LIN {X 0,Y 203.448,Z 428.589,A -85,B 0,C 180,E1 -22081.79,E2 -22081.79} C_VEL
LIN {X 0,Y 207.049,Z 418.268,A -85,B 0,C 180,E1 -22083.768,E2 -22083.768} C_VEL
LIN {X 0,Y 210.594,Z 406.82,A -85,B 0,C 180,E1 -22085.44,E2 -22085.44} C_VEL
LIN {X 0,Y 213.533,Z 394.846,A -85,B 0,C 180,E1 -22086.77,E2 -22086.77} C_VEL
LIN {X 0,Y 215.971,Z 381.541,A -85,B 0,C 180,E1 -22087.821,E2 -22087.821} C_VEL
LIN {X 0,Y 217.695,Z 368.318,A -85,B 0,C 180,E1 -22088.489,E2 -22088.489} C_VEL
LIN {X 0,Y 220.282,Z 324.105,A -85,B 0,C 180,E1 -22089.842,E2 -22089.842} C_VEL
LIN {X 0,Y 219.565,Z 319.298,A -85,B 0,C 180,E1 -22090.222,E2 -22090.222} C_VEL
LIN {X 0,Y 213.219,Z 304.183,A -85,B 0,C 180,E1 -22092.522,E2 -22092.522} C_VEL
LIN {X 0,Y 207.872,Z 293.408,A -85,B 0,C 180,E1 -22094.554,E2 -22094.554} C_VEL
LIN {X 0,Y 202.404,Z 283.572,A -85,B 0,C 180,E1 -22096.771,E2 -22096.771} C_VEL
LIN {X 0,Y 197.273,Z 275.162,A -85,B 0,C 180,E1 -22099.019,E2 -22099.019} C_VEL
LIN {X 0,Y 193.69,Z 269.753,A -85,B 0,C 180,E1 -22100.705,E2 -22100.705} C_VEL
LIN {X 0,Y 190.17,Z 264.45,A -85,B 0,C 180,E1 -22102.496,E2 -22102.496} C_VEL
LIN {X 0,Y 187.207,Z 260.568,A -85,B 0,C 180,E1 -22104.085,E2 -22104.085} C_VEL
LIN {X 0,Y 186.277,Z 258.764,A -85,B 0,C 180,E1 -22104.71,E2 -22104.71} C_VEL
LIN {X 0,Y 185.559,Z 256.36,A -85,B 0,C 180,E1 -22107.046,E2 -22107.046} C_VEL
LIN {X 0,Y 185.548,Z 256.361,A -85,B 0,C 180,E1 -22110.595,E2 -22110.595} C_VEL
LIN {X 0,Y 185.581,Z 256.359,A -85,B 0,C 180,E1 -22115.382,E2 -22115.382} C_VEL
LIN {X 0,Y 185.635,Z 256.363,A -85,B 0,C 180,E1 -22121.171,E2 -22121.171} C_VEL
LIN {X 0,Y 185.673,Z 256.35,A -85,B 0,C 180,E1 -22124.636,E2 -22124.636} C_VEL
LIN {X 0,Y 185.925,Z 256.316,A -85,B 0,C 180,E1 -22129.359,E2 -22129.359} C_VEL
LIN {X 0,Y 185.958,Z 256.306,A -85,B 0,C 180,E1 -22133.49,E2 -22133.49} C_VEL
LIN {X 0,Y 186.203,Z 256.274,A -85,B 0,C 180,E1 -22137.837,E2 -22137.837} C_VEL
LIN {X 0,Y 186.405,Z 256.262,A -85,B 0,C 180,E1 -22140,E2 -22140} C_VEL
LIN {X 0,Y 185.909,Z 256.317,A -85,B 0,C 180,E1 -22144.336,E2 -22144.336} C_VEL
LIN {X 0,Y 185.976,Z 256.304,A -85,B 0,C 180,E1 -22148.694,E2 -22148.694} C_VEL
LIN {X 0,Y 185.724,Z 256.336,A -85,B 0,C 180,E1 -22153.124,E2 -22153.124} C_VEL
LIN {X 0,Y 185.688,Z 256.34,A -85,B 0,C 180,E1 -22157.625,E2 -22157.625} C_VEL
LIN {X 0,Y 185.597,Z 256.352,A -85,B 0,C 180,E1 -22162.252,E2 -22162.252} C_VEL
LIN {X 0,Y 185.564,Z 256.36,A -85,B 0,C 180,E1 -22167.032,E2 -22167.032} C_VEL
LIN {X 0,Y 185.607,Z 256.374,A -85,B 0,C 180,E1 -22169.284,E2 -22169.284} C_VEL
LIN {X 0,Y 186.334,Z 258.759,A -85,B 0,C 180,E1 -22169.804,E2 -22169.804} C_VEL
LIN {X 0,Y 188.069,Z 260.918,A -85,B 0,C 180,E1 -22170.763,E2 -22170.763} C_VEL
LIN {X 0,Y 189.675,Z 262.213,A -85,B 0,C 180,E1 -22171.569,E2 -22171.569} C_VEL
LIN {X 0,Y 191.536,Z 265.32,A -85,B 0,C 180,E1 -22172.568,E2 -22172.568} C_VEL
LIN {X 0,Y 193.597,Z 267.452,A -85,B 0,C 180,E1 -22173.544,E2 -22173.544} C_VEL
LIN {X 0,Y 196.036,Z 270.879,A -85,B 0,C 180,E1 -22174.698,E2 -22174.698} C_VEL
LIN {X 0,Y 197.873,Z 273.45,A -85,B 0,C 180,E1 -22175.528,E2 -22175.528} C_VEL
LIN {X 0,Y 200.738,Z 277.395,A -85,B 0,C 180,E1 -22176.761,E2 -22176.761} C_VEL
LIN {X 0,Y 206.923,Z 286.536,A -85,B 0,C 180,E1 -22179.242,E2 -22179.242} C_VEL
LIN {X 0,Y 210.932,Z 293.337,A -85,B 0,C 180,E1 -22180.757,E2 -22180.757} C_VEL
LIN {X 0,Y 217.361,Z 306.275,A -85,B 0,C 180,E1 -22183.082,E2 -22183.082} C_VEL
LIN {X 0,Y 220.832,Z 314.289,A -85,B 0,C 180,E1 -22184.29,E2 -22184.29} C_VEL
LIN {X 0,Y 218.061,Z 360.113,A -85,B 0,C 180,E1 -22185.691,E2 -22185.691} C_VEL
LIN {X 0,Y 216.493,Z 373.353,A -85,B 0,C 180,E1 -22186.429,E2 -22186.429} C_VEL
LIN {X 0,Y 214.306,Z 385.674,A -85,B 0,C 180,E1 -22187.438,E2 -22187.438} C_VEL
LIN {X 0,Y 211.711,Z 396.969,A -85,B 0,C 180,E1 -22188.717,E2 -22188.717} C_VEL
LIN {X 0,Y 208.24,Z 408.631,A -85,B 0,C 180,E1 -22190.43,E2 -22190.43} C_VEL
LIN {X 0,Y 204.695,Z 419.107,A -85,B 0,C 180,E1 -22192.452,E2 -22192.452} C_VEL
LIN {X 0,Y 200.989,Z 428.49,A -85,B 0,C 180,E1 -22194.763,E2 -22194.763} C_VEL
LIN {X 0,Y 197.612,Z 436.177,A -85,B 0,C 180,E1 -22197.155,E2 -22197.155} C_VEL
LIN {X 0,Y 193.935,Z 444.033,A -85,B 0,C 180,E1 -22200.298,E2 -22200.298} C_VEL
LIN {X 0,Y 190.616,Z 450.593,A -85,B 0,C 180,E1 -22203.74,E2 -22203.74} C_VEL
LIN {X 0,Y 188.133,Z 455.122,A -85,B 0,C 180,E1 -22206.906,E2 -22206.906} C_VEL
LIN {X 0,Y 185.771,Z 459.292,A -85,B 0,C 180,E1 -22211.049,E2 -22211.049} C_VEL
LIN {X 0,Y 184.359,Z 461.532,A -85,B 0,C 180,E1 -22214.523,E2 -22214.523} C_VEL
LIN {X 0,Y 183.67,Z 462.424,A -85,B 0,C 180,E1 -22216.727,E2 -22216.727} C_VEL
LIN {X 0,Y 183.286,Z 462.899,A -85,B 0,C 180,E1 -22218.947,E2 -22218.947} C_VEL
LIN {X 0,Y 183.106,Z 462.953,A -85,B 0,C 180,E1 -22221.168,E2 -22221.168} C_VEL
LIN {X 0,Y 183.082,Z 462.624,A -85,B 0,C 180,E1 -22223.387,E2 -22223.387} C_VEL
LIN {X 0,Y 183.132,Z 461.645,A -85,B 0,C 180,E1 -22226.201,E2 -22226.201} C_VEL
LIN {X 0,Y 183.433,Z 459.249,A -85,B 0,C 180,E1 -22230,E2 -22230} C_VEL
LIN {X 0,Y 184.027,Z 456.15,A -85,B 0,C 180,E1 -22233.284,E2 -22233.284} C_VEL
LIN {X 0,Y 184.978,Z 452.007,A -85,B 0,C 180,E1 -22236.545,E2 -22236.545} C_VEL
LIN {X 0,Y 186.753,Z 445.691,A -85,B 0,C 180,E1 -22240.297,E2 -22240.297} C_VEL
LIN {X 0,Y 188.757,Z 438.816,A -85,B 0,C 180,E1 -22243.456,E2 -22243.456} C_VEL
LIN {X 0,Y 191.319,Z 430.194,A -85,B 0,C 180,E1 -22246.54,E2 -22246.54} C_VEL
LIN {X 0,Y 193.755,Z 421.37,A -85,B 0,C 180,E1 -22249.054,E2 -22249.054} C_VEL
LIN {X 0,Y 196.263,Z 411.56,A -85,B 0,C 180,E1 -22251.285,E2 -22251.285} C_VEL
LIN {X 0,Y 198.602,Z 401.054,A -85,B 0,C 180,E1 -22253.184,E2 -22253.184} C_VEL
LIN {X 0,Y 200.825,Z 389.158,A -85,B 0,C 180,E1 -22254.831,E2 -22254.831} C_VEL
LIN {X 0,Y 202.636,Z 376.778,A -85,B 0,C 180,E1 -22256.106,E2 -22256.106} C_VEL
LIN {X 0,Y 203.926,Z 363.965,A -85,B 0,C 180,E1 -22257.031,E2 -22257.031} C_VEL
LIN {X 0,Y 204.857,Z 349.414,A -85,B 0,C 180,E1 -22257.622,E2 -22257.622} C_VEL
LIN {X 0,Y 207.063,Z 299.532,A -85,B 0,C 180,E1 -22259.251,E2 -22259.251} C_VEL
LIN {X 0,Y 200.953,Z 283.961,A -85,B 0,C 180,E1 -22261.036,E2 -22261.036} C_VEL
LIN {X 0,Y 195.353,Z 273.341,A -85,B 0,C 180,E1 -22262.644,E2 -22262.644} C_VEL
LIN {X 0,Y 189.717,Z 264.038,A -85,B 0,C 180,E1 -22264.328,E2 -22264.328} C_VEL
LIN {X 0,Y 187.441,Z 260.424,A -85,B 0,C 180,E1 -22265.042,E2 -22265.042} C_VEL
LIN {X 0,Y 185.812,Z 257.687,A -85,B 0,C 180,E1 -22265.575,E2 -22265.575} C_VEL
LIN {X 0,Y 185.526,Z 256.374,A -85,B 0,C 180,E1 -22265.765,E2 -22265.765} C_VEL
LIN {X 0,Y 185.473,Z 256.381,A -85,B 0,C 180,E1 -22270.725,E2 -22270.725} C_VEL
LIN {X 0,Y 185.463,Z 256.382,A -85,B 0,C 180,E1 -22276.054,E2 -22276.054} C_VEL
LIN {X 0,Y 185.47,Z 256.382,A -85,B 0,C 180,E1 -22279.895,E2 -22279.895} C_VEL
LIN {X 0,Y 185.508,Z 256.377,A -85,B 0,C 180,E1 -22282.711,E2 -22282.711} C_VEL
LIN {X 0,Y 185.543,Z 256.343,A -85,B 0,C 180,E1 -22287.974,E2 -22287.974} C_VEL
LIN {X 0,Y 185.582,Z 256.359,A -85,B 0,C 180,E1 -22290.576,E2 -22290.576} C_VEL
LIN {X 0,Y 185.589,Z 256.348,A -85,B 0,C 180,E1 -22295.382,E2 -22295.382} C_VEL
LIN {X 0,Y 185.676,Z 256.346,A -85,B 0,C 180,E1 -22301.133,E2 -22301.133} C_VEL
LIN {X 0,Y 185.696,Z 256.345,A -85,B 0,C 180,E1 -22304.637,E2 -22304.637} C_VEL
LIN {X 0,Y 185.889,Z 256.288,A -85,B 0,C 180,E1 -22309.419,E2 -22309.419} C_VEL
LIN {X 0,Y 185.938,Z 256.318,A -85,B 0,C 180,E1 -22313.489,E2 -22313.489} C_VEL
LIN {X 0,Y 186.204,Z 256.277,A -85,B 0,C 180,E1 -22317.837,E2 -22317.837} C_VEL
LIN {X 0,Y 186.405,Z 256.262,A -85,B 0,C 180,E1 -22320,E2 -22320} C_VEL
LIN {X 0,Y 185.923,Z 256.315,A -85,B 0,C 180,E1 -22324.336,E2 -22324.336} C_VEL
LIN {X 0,Y 186.03,Z 256.307,A -85,B 0,C 180,E1 -22328.691,E2 -22328.691} C_VEL
LIN {X 0,Y 185.726,Z 256.342,A -85,B 0,C 180,E1 -22333.123,E2 -22333.123} C_VEL
LIN {X 0,Y 185.657,Z 256.347,A -85,B 0,C 180,E1 -22337.628,E2 -22337.628} C_VEL
LIN {X 0,Y 185.571,Z 256.37,A -85,B 0,C 180,E1 -22342.254,E2 -22342.254} C_VEL
LIN {X 0,Y 185.577,Z 256.357,A -85,B 0,C 180,E1 -22344.646,E2 -22344.646} C_VEL
LIN {X 0,Y 185.544,Z 256.367,A -85,B 0,C 180,E1 -22349.499,E2 -22349.499} C_VEL
LIN {X 0,Y 185.497,Z 256.372,A -85,B 0,C 180,E1 -22354.632,E2 -22354.632} C_VEL
LIN {X 0,Y 185.501,Z 256.378,A -85,B 0,C 180,E1 -22357.314,E2 -22357.314} C_VEL
LIN {X 0,Y 185.464,Z 256.384,A -85,B 0,C 180,E1 -22360.722,E2 -22360.722} C_VEL
LIN {X 0,Y 185.47,Z 256.406,A -85,B 0,C 180,E1 -22366.098,E2 -22366.098} C_VEL
LIN {X 0,Y 186.5,Z 260.261,A -85,B 0,C 180,E1 -22368.365,E2 -22368.365} C_VEL
LIN {X 0,Y 188.973,Z 264.686,A -85,B 0,C 180,E1 -22369.172,E2 -22369.172} C_VEL
LIN {X 0,Y 195.749,Z 278.235,A -85,B 0,C 180,E1 -22371.304,E2 -22371.304} C_VEL
LIN {X 0,Y 202.24,Z 293.675,A -85,B 0,C 180,E1 -22373.268,E2 -22373.268} C_VEL
LIN {X 0,Y 204.621,Z 300.449,A -85,B 0,C 180,E1 -22373.993,E2 -22373.993} C_VEL
LIN {X 0,Y 206.416,Z 317.831,A -85,B 0,C 180,E1 -22375.02,E2 -22375.02} C_VEL
LIN {X 0,Y 206.011,Z 326.955,A -85,B 0,C 180,E1 -22375.317,E2 -22375.317} C_VEL
LIN {X 0,Y 205.217,Z 332.797,A -85,B 0,C 180,E1 -22375.416,E2 -22375.416} C_VEL
LIN {X 0,Y 199.436,Z 351.769,A -85,B 0,C 180,E1 -22375.178,E2 -22375.178} C_VEL
LIN {X 0,Y 198.574,Z 357.613,A -85,B 0,C 180,E1 -22375.267,E2 -22375.267} C_VEL
LIN {X 0,Y 197.647,Z 372.415,A -85,B 0,C 180,E1 -22375.864,E2 -22375.864} C_VEL
LIN {X 0,Y 196.156,Z 385.164,A -85,B 0,C 180,E1 -22376.727,E2 -22376.727} C_VEL
LIN {X 0,Y 194.021,Z 397.941,A -85,B 0,C 180,E1 -22378.011,E2 -22378.011} C_VEL
LIN {X 0,Y 191.532,Z 410.148,A -85,B 0,C 180,E1 -22379.7,E2 -22379.7} C_VEL
LIN {X 0,Y 188.837,Z 421.006,A -85,B 0,C 180,E1 -22381.672,E2 -22381.672} C_VEL
LIN {X 0,Y 185.792,Z 431.841,A -85,B 0,C 180,E1 -22384.214,E2 -22384.214} C_VEL
LIN {X 0,Y 183.265,Z 441.005,A -85,B 0,C 180,E1 -22386.981,E2 -22386.981} C_VEL
LIN {X 0,Y 181.313,Z 447.926,A -85,B 0,C 180,E1 -22389.583,E2 -22389.583} C_VEL
LIN {X 0,Y 179.202,Z 455.049,A -85,B 0,C 180,E1 -22392.894,E2 -22392.894} C_VEL
LIN {X 0,Y 177.601,Z 460.726,A -85,B 0,C 180,E1 -22396.265,E2 -22396.265} C_VEL
LIN {X 0,Y 176.675,Z 465.196,A -85,B 0,C 180,E1 -22399.688,E2 -22399.688} C_VEL
LIN {X 0,Y 176.137,Z 468.572,A -85,B 0,C 180,E1 -22403.125,E2 -22403.125} C_VEL
LIN {X 0,Y 175.995,Z 471.007,A -85,B 0,C 180,E1 -22406.681,E2 -22406.681} C_VEL
LIN {X 0,Y 176.092,Z 472.381,A -85,B 0,C 180,E1 -22410,E2 -22410} C_VEL
LIN {X 0,Y 175.97,Z 472.854,A -85,B 0,C 180,E1 -22413.176,E2 -22413.176} C_VEL
LIN {X 0,Y 176.141,Z 472.465,A -85,B 0,C 180,E1 -22416.875,E2 -22416.875} C_VEL
LIN {X 0,Y 176.481,Z 471.725,A -85,B 0,C 180,E1 -22419.166,E2 -22419.166} C_VEL
LIN {X 0,Y 177.064,Z 470.558,A -85,B 0,C 180,E1 -22421.447,E2 -22421.447} C_VEL
LIN {X 0,Y 177.887,Z 468.974,A -85,B 0,C 180,E1 -22423.713,E2 -22423.713} C_VEL
LIN {X 0,Y 179.541,Z 465.81,A -85,B 0,C 180,E1 -22427.073,E2 -22427.073} C_VEL
LIN {X 0,Y 181.936,Z 461.603,A -85,B 0,C 180,E1 -22430.344,E2 -22430.344} C_VEL
LIN {X 0,Y 185.407,Z 455.225,A -85,B 0,C 180,E1 -22434.047,E2 -22434.047} C_VEL
LIN {X 0,Y 188.77,Z 448.292,A -85,B 0,C 180,E1 -22437.134,E2 -22437.134} C_VEL
LIN {X 0,Y 192.793,Z 439.621,A -85,B 0,C 180,E1 -22440.082,E2 -22440.082} C_VEL
LIN {X 0,Y 196.671,Z 430.752,A -85,B 0,C 180,E1 -22442.413,E2 -22442.413} C_VEL
LIN {X 0,Y 200.782,Z 419.841,A -85,B 0,C 180,E1 -22444.667,E2 -22444.667} C_VEL
LIN {X 0,Y 204.401,Z 408.803,A -85,B 0,C 180,E1 -22446.378,E2 -22446.378} C_VEL
LIN {X 0,Y 207.665,Z 396.448,A -85,B 0,C 180,E1 -22447.836,E2 -22447.836} C_VEL
LIN {X 0,Y 210.073,Z 384.716,A -85,B 0,C 180,E1 -22448.85,E2 -22448.85} C_VEL
LIN {X 0,Y 211.952,Z 371.86,A -85,B 0,C 180,E1 -22449.599,E2 -22449.599} C_VEL
LIN {X 0,Y 213.178,Z 357.263,A -85,B 0,C 180,E1 -22450.1,E2 -22450.1} C_VEL
LIN {X 0,Y 214.965,Z 324.362,A -85,B 0,C 180,E1 -22451.136,E2 -22451.136} C_VEL
LIN {X 0,Y 214.444,Z 321.886,A -85,B 0,C 180,E1 -22451.382,E2 -22451.382} C_VEL
LIN {X 0,Y 208.578,Z 307.84,A -85,B 0,C 180,E1 -22453.637,E2 -22453.637} C_VEL
LIN {X 0,Y 203.693,Z 297.749,A -85,B 0,C 180,E1 -22455.61,E2 -22455.61} C_VEL
LIN {X 0,Y 198.733,Z 288.663,A -85,B 0,C 180,E1 -22457.736,E2 -22457.736} C_VEL
LIN {X 0,Y 193.493,Z 279.929,A -85,B 0,C 180,E1 -22460.167,E2 -22460.167} C_VEL
LIN {X 0,Y 190.645,Z 275.459,A -85,B 0,C 180,E1 -22461.59,E2 -22461.59} C_VEL
LIN {X 0,Y 186.999,Z 269.999,A -85,B 0,C 180,E1 -22463.539,E2 -22463.539} C_VEL
LIN {X 0,Y 183.891,Z 265.461,A -85,B 0,C 180,E1 -22465.339,E2 -22465.339} C_VEL
LIN {X 0,Y 179.125,Z 259.472,A -85,B 0,C 180,E1 -22468.347,E2 -22468.347} C_VEL
LIN {X 0,Y 178.697,Z 258.346,A -85,B 0,C 180,E1 -22468.758,E2 -22468.758} C_VEL
LIN {X 0,Y 178.482,Z 257.241,A -85,B 0,C 180,E1 -22470.03,E2 -22470.03} C_VEL
LIN {X 0,Y 178.516,Z 257.237,A -85,B 0,C 180,E1 -22474.889,E2 -22474.889} C_VEL
LIN {X 0,Y 178.591,Z 257.239,A -85,B 0,C 180,E1 -22480.814,E2 -22480.814} C_VEL
LIN {X 0,Y 178.651,Z 257.227,A -85,B 0,C 180,E1 -22486.347,E2 -22486.347} C_VEL
LIN {X 0,Y 178.961,Z 257.19,A -85,B 0,C 180,E1 -22490.962,E2 -22490.962} C_VEL
LIN {X 0,Y 179.149,Z 257.153,A -85,B 0,C 180,E1 -22497.752,E2 -22497.752} C_VEL
LIN {X 0,Y 179.368,Z 257.138,A -85,B 0,C 180,E1 -22500,E2 -22500} C_VEL
LIN {X 0,Y 178.857,Z 257.196,A -85,B 0,C 180,E1 -22504.508,E2 -22504.508} C_VEL
LIN {X 0,Y 178.906,Z 257.186,A -85,B 0,C 180,E1 -22509.041,E2 -22509.041} C_VEL
LIN {X 0,Y 178.653,Z 257.216,A -85,B 0,C 180,E1 -22513.653,E2 -22513.653} C_VEL
LIN {X 0,Y 178.624,Z 257.223,A -85,B 0,C 180,E1 -22519.216,E2 -22519.216} C_VEL
LIN {X 0,Y 178.534,Z 257.239,A -85,B 0,C 180,E1 -22525.274,E2 -22525.274} C_VEL
LIN {X 0,Y 178.539,Z 257.332,A -85,B 0,C 180,E1 -22525.562,E2 -22525.562} C_VEL
LIN {X 0,Y 179.259,Z 259.662,A -85,B 0,C 180,E1 -22526.172,E2 -22526.172} C_VEL
LIN {X 0,Y 181.191,Z 261.941,A -85,B 0,C 180,E1 -22527.427,E2 -22527.427} C_VEL
LIN {X 0,Y 182.827,Z 263.049,A -85,B 0,C 180,E1 -22528.373,E2 -22528.373} C_VEL
LIN {X 0,Y 184.655,Z 266.207,A -85,B 0,C 180,E1 -22529.518,E2 -22529.518} C_VEL
LIN {X 0,Y 186.908,Z 268.442,A -85,B 0,C 180,E1 -22530.74,E2 -22530.74} C_VEL
LIN {X 0,Y 189.389,Z 271.993,A -85,B 0,C 180,E1 -22532.082,E2 -22532.082} C_VEL
LIN {X 0,Y 190.753,Z 273.562,A -85,B 0,C 180,E1 -22532.762,E2 -22532.762} C_VEL
LIN {X 0,Y 194.542,Z 278.861,A -85,B 0,C 180,E1 -22534.601,E2 -22534.601} C_VEL
LIN {X 0,Y 199.477,Z 285.887,A -85,B 0,C 180,E1 -22536.795,E2 -22536.795} C_VEL
LIN {X 0,Y 205.61,Z 295.649,A -85,B 0,C 180,E1 -22539.303,E2 -22539.303} C_VEL
LIN {X 0,Y 211.796,Z 308.073,A -85,B 0,C 180,E1 -22541.701,E2 -22541.701} C_VEL
LIN {X 0,Y 215.496,Z 316.487,A -85,B 0,C 180,E1 -22543.069,E2 -22543.069} C_VEL
LIN {X 0,Y 212.733,Z 360.615,A -85,B 0,C 180,E1 -22544.451,E2 -22544.451} C_VEL
LIN {X 0,Y 211.091,Z 373.864,A -85,B 0,C 180,E1 -22545.206,E2 -22545.206} C_VEL
LIN {X 0,Y 208.85,Z 385.963,A -85,B 0,C 180,E1 -22546.215,E2 -22546.215} C_VEL
LIN {X 0,Y 205.925,Z 398.03,A -85,B 0,C 180,E1 -22547.62,E2 -22547.62} C_VEL
LIN {X 0,Y 202.321,Z 409.533,A -85,B 0,C 180,E1 -22549.36,E2 -22549.36} C_VEL
LIN {X 0,Y 198.799,Z 419.507,A -85,B 0,C 180,E1 -22551.344,E2 -22551.344} C_VEL
LIN {X 0,Y 195.169,Z 428.309,A -85,B 0,C 180,E1 -22553.547,E2 -22553.547} C_VEL
LIN {X 0,Y 191.584,Z 436.061,A -85,B 0,C 180,E1 -22555.984,E2 -22555.984} C_VEL
LIN {X 0,Y 187.589,Z 444.231,A -85,B 0,C 180,E1 -22559.329,E2 -22559.329} C_VEL
LIN {X 0,Y 184.177,Z 450.592,A -85,B 0,C 180,E1 -22562.748,E2 -22562.748} C_VEL
LIN {X 0,Y 181.538,Z 455.17,A -85,B 0,C 180,E1 -22566.015,E2 -22566.015} C_VEL
LIN {X 0,Y 179.44,Z 458.636,A -85,B 0,C 180,E1 -22569.36,E2 -22569.36} C_VEL
LIN {X 0,Y 178.349,Z 460.36,A -85,B 0,C 180,E1 -22571.624,E2 -22571.624} C_VEL
LIN {X 0,Y 177.433,Z 461.666,A -85,B 0,C 180,E1 -22573.903,E2 -22573.903} C_VEL
LIN {X 0,Y 176.248,Z 463.086,A -85,B 0,C 180,E1 -22578.499,E2 -22578.499} C_VEL
LIN {X 0,Y 176.025,Z 463.16,A -85,B 0,C 180,E1 -22580.81,E2 -22580.81} C_VEL
LIN {X 0,Y 175.973,Z 462.849,A -85,B 0,C 180,E1 -22583.119,E2 -22583.119} C_VEL
LIN {X 0,Y 176.044,Z 461.72,A -85,B 0,C 180,E1 -22586.426,E2 -22586.426} C_VEL
LIN {X 0,Y 176.344,Z 459.547,A -85,B 0,C 180,E1 -22590,E2 -22590} C_VEL
LIN {X 0,Y 176.97,Z 456.487,A -85,B 0,C 180,E1 -22593.415,E2 -22593.415} C_VEL
LIN {X 0,Y 177.957,Z 452.386,A -85,B 0,C 180,E1 -22596.804,E2 -22596.804} C_VEL
LIN {X 0,Y 179.796,Z 446.116,A -85,B 0,C 180,E1 -22600.7,E2 -22600.7} C_VEL
LIN {X 0,Y 181.895,Z 439.295,A -85,B 0,C 180,E1 -22603.974,E2 -22603.974} C_VEL
LIN {X 0,Y 184.563,Z 430.76,A -85,B 0,C 180,E1 -22607.164,E2 -22607.164} C_VEL
LIN {X 0,Y 187.088,Z 422.011,A -85,B 0,C 180,E1 -22609.76,E2 -22609.76} C_VEL
LIN {X 0,Y 189.92,Z 411.473,A -85,B 0,C 180,E1 -22612.233,E2 -22612.233} C_VEL
LIN {X 0,Y 192.466,Z 400.411,A -85,B 0,C 180,E1 -22614.255,E2 -22614.255} C_VEL
LIN {X 0,Y 194.807,Z 388.28,A -85,B 0,C 180,E1 -22615.94,E2 -22615.94} C_VEL
LIN {X 0,Y 196.662,Z 375.572,A -85,B 0,C 180,E1 -22617.25,E2 -22617.25} C_VEL
LIN {X 0,Y 197.989,Z 362.526,A -85,B 0,C 180,E1 -22618.147,E2 -22618.147} C_VEL
LIN {X 0,Y 199.089,Z 343.717,A -85,B 0,C 180,E1 -22618.867,E2 -22618.867} C_VEL
LIN {X 0,Y 201.058,Z 301.314,A -85,B 0,C 180,E1 -22620.281,E2 -22620.281} C_VEL
LIN {X 0,Y 195.021,Z 286.063,A -85,B 0,C 180,E1 -22622.148,E2 -22622.148} C_VEL
LIN {X 0,Y 187.68,Z 272.688,A -85,B 0,C 180,E1 -22624.399,E2 -22624.399} C_VEL
LIN {X 0,Y 180.717,Z 261.583,A -85,B 0,C 180,E1 -22626.697,E2 -22626.697} C_VEL
LIN {X 0,Y 179.059,Z 259.332,A -85,B 0,C 180,E1 -22627.262,E2 -22627.262} C_VEL
LIN {X 0,Y 178.448,Z 257.256,A -85,B 0,C 180,E1 -22627.622,E2 -22627.622} C_VEL
LIN {X 0,Y 178.4,Z 257.26,A -85,B 0,C 180,E1 -22632.044,E2 -22632.044} C_VEL
LIN {X 0,Y 178.396,Z 257.262,A -85,B 0,C 180,E1 -22635.163,E2 -22635.163} C_VEL
LIN {X 0,Y 178.405,Z 257.261,A -85,B 0,C 180,E1 -22638.458,E2 -22638.458} C_VEL
LIN {X 0,Y 178.424,Z 257.259,A -85,B 0,C 180,E1 -22643.783,E2 -22643.783} C_VEL
LIN {X 0,Y 178.487,Z 257.226,A -85,B 0,C 180,E1 -22646.546,E2 -22646.546} C_VEL
LIN {X 0,Y 178.523,Z 257.234,A -85,B 0,C 180,E1 -22650.007,E2 -22650.007} C_VEL
LIN {X 0,Y 178.536,Z 257.232,A -85,B 0,C 180,E1 -22654.875,E2 -22654.875} C_VEL
LIN {X 0,Y 178.624,Z 257.22,A -85,B 0,C 180,E1 -22660.783,E2 -22660.783} C_VEL
LIN {X 0,Y 178.659,Z 257.205,A -85,B 0,C 180,E1 -22666.348,E2 -22666.348} C_VEL
LIN {X 0,Y 178.906,Z 257.169,A -85,B 0,C 180,E1 -22670.959,E2 -22670.959} C_VEL
LIN {X 0,Y 179.15,Z 257.156,A -85,B 0,C 180,E1 -22677.751,E2 -22677.751} C_VEL
LIN {X 0,Y 179.368,Z 257.138,A -85,B 0,C 180,E1 -22680,E2 -22680} C_VEL
LIN {X 0,Y 178.872,Z 257.193,A -85,B 0,C 180,E1 -22684.507,E2 -22684.507} C_VEL
LIN {X 0,Y 178.978,Z 257.184,A -85,B 0,C 180,E1 -22689.037,E2 -22689.037} C_VEL
LIN {X 0,Y 178.65,Z 257.228,A -85,B 0,C 180,E1 -22693.653,E2 -22693.653} C_VEL
LIN {X 0,Y 178.59,Z 257.225,A -85,B 0,C 180,E1 -22699.185,E2 -22699.185} C_VEL
LIN {X 0,Y 178.516,Z 257.236,A -85,B 0,C 180,E1 -22705.111,E2 -22705.111} C_VEL
LIN {X 0,Y 178.46,Z 257.247,A -85,B 0,C 180,E1 -22710.794,E2 -22710.794} C_VEL
LIN {X 0,Y 178.483,Z 257.247,A -85,B 0,C 180,E1 -22714.218,E2 -22714.218} C_VEL
LIN {X 0,Y 178.389,Z 257.259,A -85,B 0,C 180,E1 -22719.076,E2 -22719.076} C_VEL
LIN {X 0,Y 178.407,Z 257.26,A -85,B 0,C 180,E1 -22724.127,E2 -22724.127} C_VEL
LIN {X 0,Y 178.403,Z 257.409,A -85,B 0,C 180,E1 -22724.839,E2 -22724.839} C_VEL
LIN {X 0,Y 179.125,Z 260.011,A -85,B 0,C 180,E1 -22726.438,E2 -22726.438} C_VEL
LIN {X 0,Y 181.613,Z 264.393,A -85,B 0,C 180,E1 -22727.329,E2 -22727.329} C_VEL
LIN {X 0,Y 187.138,Z 274.745,A -85,B 0,C 180,E1 -22729.215,E2 -22729.215} C_VEL
LIN {X 0,Y 192.627,Z 286.531,A -85,B 0,C 180,E1 -22731.008,E2 -22731.008} C_VEL
LIN {X 0,Y 198.667,Z 302.088,A -85,B 0,C 180,E1 -22732.936,E2 -22732.936} C_VEL
LIN {X 0,Y 200.401,Z 318.499,A -85,B 0,C 180,E1 -22733.964,E2 -22733.964} C_VEL
LIN {X 0,Y 198.574,Z 357.613,A -85,B 0,C 180,E1 -22735.267,E2 -22735.267} C_VEL
LIN {X 0,Y 197.631,Z 363.46,A -85,B 0,C 180,E1 -22735.349,E2 -22735.349} C_VEL
LIN {X 0,Y 192.837,Z 376.555,A -85,B 0,C 180,E1 -22735.319,E2 -22735.319} C_VEL
LIN {X 0,Y 190.175,Z 384.482,A -85,B 0,C 180,E1 -22735.601,E2 -22735.601} C_VEL
LIN {X 0,Y 189.634,Z 387.751,A -85,B 0,C 180,E1 -22735.889,E2 -22735.889} C_VEL
LIN {X 0,Y 187.641,Z 398.984,A -85,B 0,C 180,E1 -22737.106,E2 -22737.106} C_VEL
LIN {X 0,Y 185.063,Z 410.888,A -85,B 0,C 180,E1 -22738.84,E2 -22738.84} C_VEL
LIN {X 0,Y 182.251,Z 421.541,A -85,B 0,C 180,E1 -22740.867,E2 -22740.867} C_VEL
LIN {X 0,Y 179.383,Z 431.269,A -85,B 0,C 180,E1 -22743.221,E2 -22743.221} C_VEL
LIN {X 0,Y 176.762,Z 440.313,A -85,B 0,C 180,E1 -22746.013,E2 -22746.013} C_VEL
LIN {X 0,Y 174.665,Z 447.471,A -85,B 0,C 180,E1 -22748.769,E2 -22748.769} C_VEL
LIN {X 0,Y 172.375,Z 454.654,A -85,B 0,C 180,E1 -22752.195,E2 -22752.195} C_VEL
LIN {X 0,Y 170.657,Z 460.373,A -85,B 0,C 180,E1 -22755.695,E2 -22755.695} C_VEL
LIN {X 0,Y 169.666,Z 464.88,A -85,B 0,C 180,E1 -22759.257,E2 -22759.257} C_VEL
LIN {X 0,Y 169.072,Z 468.29,A -85,B 0,C 180,E1 -22762.836,E2 -22762.836} C_VEL
LIN {X 0,Y 168.892,Z 471.011,A -85,B 0,C 180,E1 -22767.079,E2 -22767.079} C_VEL
LIN {X 0,Y 169,Z 472.151,A -85,B 0,C 180,E1 -22770,E2 -22770} C_VEL
LIN {X 0,Y 168.892,Z 472.627,A -85,B 0,C 180,E1 -22772.921,E2 -22772.921} C_VEL
LIN {X 0,Y 169.094,Z 472.291,A -85,B 0,C 180,E1 -22777.163,E2 -22777.163} C_VEL
LIN {X 0,Y 169.464,Z 471.566,A -85,B 0,C 180,E1 -22779.549,E2 -22779.549} C_VEL
LIN {X 0,Y 170.088,Z 470.43,A -85,B 0,C 180,E1 -22781.923,E2 -22781.923} C_VEL
LIN {X 0,Y 170.963,Z 468.861,A -85,B 0,C 180,E1 -22784.279,E2 -22784.279} C_VEL
LIN {X 0,Y 172.747,Z 465.731,A -85,B 0,C 180,E1 -22787.766,E2 -22787.766} C_VEL
LIN {X 0,Y 175.264,Z 461.559,A -85,B 0,C 180,E1 -22791.155,E2 -22791.155} C_VEL
LIN {X 0,Y 178.915,Z 455.22,A -85,B 0,C 180,E1 -22794.978,E2 -22794.978} C_VEL
LIN {X 0,Y 182.456,Z 448.334,A -85,B 0,C 180,E1 -22798.155,E2 -22798.155} C_VEL
LIN {X 0,Y 185.918,Z 441.315,A -85,B 0,C 180,E1 -22800.685,E2 -22800.685} C_VEL
LIN {X 0,Y 189.881,Z 432.868,A -85,B 0,C 180,E1 -22803.089,E2 -22803.089} C_VEL
LIN {X 0,Y 194.114,Z 422.447,A -85,B 0,C 180,E1 -22805.4,E2 -22805.4} C_VEL
LIN {X 0,Y 198.272,Z 410.726,A -85,B 0,C 180,E1 -22807.374,E2 -22807.374} C_VEL
LIN {X 0,Y 201.624,Z 398.996,A -85,B 0,C 180,E1 -22808.86,E2 -22808.86} C_VEL
LIN {X 0,Y 204.379,Z 386.812,A -85,B 0,C 180,E1 -22809.987,E2 -22809.987} C_VEL
LIN {X 0,Y 206.491,Z 373.856,A -85,B 0,C 180,E1 -22810.821,E2 -22810.821} C_VEL
LIN {X 0,Y 207.751,Z 361.194,A -85,B 0,C 180,E1 -22811.31,E2 -22811.31} C_VEL
LIN {X 0,Y 209.831,Z 325.699,A -85,B 0,C 180,E1 -22812.427,E2 -22812.427} C_VEL
LIN {X 0,Y 203.908,Z 311.096,A -85,B 0,C 180,E1 -22814.856,E2 -22814.856} C_VEL
LIN {X 0,Y 198.277,Z 299.46,A -85,B 0,C 180,E1 -22817.296,E2 -22817.296} C_VEL
LIN {X 0,Y 193.123,Z 290.249,A -85,B 0,C 180,E1 -22819.692,E2 -22819.692} C_VEL
LIN {X 0,Y 189.765,Z 284.6,A -85,B 0,C 180,E1 -22821.379,E2 -22821.379} C_VEL
LIN {X 0,Y 187.166,Z 280.492,A -85,B 0,C 180,E1 -22822.76,E2 -22822.76} C_VEL
LIN {X 0,Y 184.182,Z 275.82,A -85,B 0,C 180,E1 -22824.457,E2 -22824.457} C_VEL
LIN {X 0,Y 180.573,Z 270.52,A -85,B 0,C 180,E1 -22826.674,E2 -22826.674} C_VEL
LIN {X 0,Y 176.506,Z 265.148,A -85,B 0,C 180,E1 -22829.431,E2 -22829.431} C_VEL
LIN {X 0,Y 175.514,Z 263.719,A -85,B 0,C 180,E1 -22830.174,E2 -22830.174} C_VEL
LIN {X 0,Y 172.876,Z 261.666,A -85,B 0,C 180,E1 -22832.127,E2 -22832.127} C_VEL
LIN {X 0,Y 171.659,Z 259.391,A -85,B 0,C 180,E1 -22833.233,E2 -22833.233} C_VEL
LIN {X 0,Y 171.417,Z 258.123,A -85,B 0,C 180,E1 -22833.644,E2 -22833.644} C_VEL
LIN {X 0,Y 171.446,Z 258.118,A -85,B 0,C 180,E1 -22838.35,E2 -22838.35} C_VEL
LIN {X 0,Y 171.547,Z 258.117,A -85,B 0,C 180,E1 -22840.868,E2 -22840.868} C_VEL
LIN {X 0,Y 171.565,Z 258.114,A -85,B 0,C 180,E1 -22845.772,E2 -22845.772} C_VEL
LIN {X 0,Y 171.889,Z 258.073,A -85,B 0,C 180,E1 -22850.587,E2 -22850.587} C_VEL
LIN {X 0,Y 171.815,Z 258.081,A -85,B 0,C 180,E1 -22855.308,E2 -22855.308} C_VEL
LIN {X 0,Y 172.331,Z 258.014,A -85,B 0,C 180,E1 -22860,E2 -22860} C_VEL
LIN {X 0,Y 171.805,Z 258.076,A -85,B 0,C 180,E1 -22864.693,E2 -22864.693} C_VEL
LIN {X 0,Y 171.844,Z 258.067,A -85,B 0,C 180,E1 -22869.416,E2 -22869.416} C_VEL
LIN {X 0,Y 171.57,Z 258.1,A -85,B 0,C 180,E1 -22874.228,E2 -22874.228} C_VEL
LIN {X 0,Y 171.546,Z 258.107,A -85,B 0,C 180,E1 -22879.562,E2 -22879.562} C_VEL
LIN {X 0,Y 171.476,Z 258.119,A -85,B 0,C 180,E1 -22880.906,E2 -22880.906} C_VEL
LIN {X 0,Y 172.277,Z 260.684,A -85,B 0,C 180,E1 -22881.776,E2 -22881.776} C_VEL
LIN {X 0,Y 174.2,Z 262.88,A -85,B 0,C 180,E1 -22883.321,E2 -22883.321} C_VEL
LIN {X 0,Y 176.108,Z 264.163,A -85,B 0,C 180,E1 -22884.665,E2 -22884.665} C_VEL
LIN {X 0,Y 177.889,Z 267.232,A -85,B 0,C 180,E1 -22885.995,E2 -22885.995} C_VEL
LIN {X 0,Y 180.461,Z 269.643,A -85,B 0,C 180,E1 -22887.625,E2 -22887.625} C_VEL
LIN {X 0,Y 182.894,Z 273.15,A -85,B 0,C 180,E1 -22889.147,E2 -22889.147} C_VEL
LIN {X 0,Y 184.323,Z 274.72,A -85,B 0,C 180,E1 -22889.96,E2 -22889.96} C_VEL
LIN {X 0,Y 187.29,Z 278.64,A -85,B 0,C 180,E1 -22891.598,E2 -22891.598} C_VEL
LIN {X 0,Y 192.017,Z 285.354,A -85,B 0,C 180,E1 -22894.008,E2 -22894.008} C_VEL
LIN {X 0,Y 196.467,Z 291.951,A -85,B 0,C 180,E1 -22896.076,E2 -22896.076} C_VEL
LIN {X 0,Y 201.618,Z 300.255,A -85,B 0,C 180,E1 -22898.286,E2 -22898.286} C_VEL
LIN {X 0,Y 207.614,Z 312.601,A -85,B 0,C 180,E1 -22900.746,E2 -22900.746} C_VEL
LIN {X 0,Y 210.286,Z 318.792,A -85,B 0,C 180,E1 -22901.795,E2 -22901.795} C_VEL
LIN {X 0,Y 207.563,Z 360.704,A -85,B 0,C 180,E1 -22903.129,E2 -22903.129} C_VEL
LIN {X 0,Y 205.915,Z 373.674,A -85,B 0,C 180,E1 -22903.873,E2 -22903.873} C_VEL
LIN {X 0,Y 203.502,Z 386.263,A -85,B 0,C 180,E1 -22904.93,E2 -22904.93} C_VEL
LIN {X 0,Y 200.683,Z 397.501,A -85,B 0,C 180,E1 -22906.239,E2 -22906.239} C_VEL
LIN {X 0,Y 196.948,Z 409.135,A -85,B 0,C 180,E1 -22908.004,E2 -22908.004} C_VEL
LIN {X 0,Y 192.98,Z 419.881,A -85,B 0,C 180,E1 -22910.16,E2 -22910.16} C_VEL
LIN {X 0,Y 189.46,Z 428.113,A -85,B 0,C 180,E1 -22912.261,E2 -22912.261} C_VEL
LIN {X 0,Y 185.661,Z 435.942,A -85,B 0,C 180,E1 -22914.741,E2 -22914.741} C_VEL
LIN {X 0,Y 181.816,Z 443.447,A -85,B 0,C 180,E1 -22917.823,E2 -22917.823} C_VEL
LIN {X 0,Y 177.793,Z 450.582,A -85,B 0,C 180,E1 -22921.683,E2 -22921.683} C_VEL
LIN {X 0,Y 174.971,Z 455.21,A -85,B 0,C 180,E1 -22925.055,E2 -22925.055} C_VEL
LIN {X 0,Y 172.724,Z 458.714,A -85,B 0,C 180,E1 -22928.518,E2 -22928.518} C_VEL
LIN {X 0,Y 171.535,Z 460.475,A -85,B 0,C 180,E1 -22930.867,E2 -22930.867} C_VEL
LIN {X 0,Y 169.751,Z 462.728,A -85,B 0,C 180,E1 -22935.616,E2 -22935.616} C_VEL
LIN {X 0,Y 169.235,Z 463.265,A -85,B 0,C 180,E1 -22938.016,E2 -22938.016} C_VEL
LIN {X 0,Y 168.966,Z 463.367,A -85,B 0,C 180,E1 -22940.423,E2 -22940.423} C_VEL
LIN {X 0,Y 168.882,Z 463.075,A -85,B 0,C 180,E1 -22942.828,E2 -22942.828} C_VEL
LIN {X 0,Y 168.96,Z 461.798,A -85,B 0,C 180,E1 -22946.663,E2 -22946.663} C_VEL
LIN {X 0,Y 169.238,Z 459.846,A -85,B 0,C 180,E1 -22950,E2 -22950} C_VEL
LIN {X 0,Y 169.915,Z 456.824,A -85,B 0,C 180,E1 -22953.557,E2 -22953.557} C_VEL
LIN {X 0,Y 170.941,Z 452.766,A -85,B 0,C 180,E1 -22957.085,E2 -22957.085} C_VEL
LIN {X 0,Y 172.852,Z 446.542,A -85,B 0,C 180,E1 -22961.135,E2 -22961.135} C_VEL
LIN {X 0,Y 175.051,Z 439.771,A -85,B 0,C 180,E1 -22964.532,E2 -22964.532} C_VEL
LIN {X 0,Y 177.832,Z 431.326,A -85,B 0,C 180,E1 -22967.835,E2 -22967.835} C_VEL
LIN {X 0,Y 180.869,Z 421.31,A -85,B 0,C 180,E1 -22970.88,E2 -22970.88} C_VEL
LIN {X 0,Y 183.447,Z 411.995,A -85,B 0,C 180,E1 -22973.116,E2 -22973.116} C_VEL
LIN {X 0,Y 186.042,Z 401.321,A -85,B 0,C 180,E1 -22975.15,E2 -22975.15} C_VEL
LIN {X 0,Y 188.476,Z 389.383,A -85,B 0,C 180,E1 -22976.88,E2 -22976.88} C_VEL
LIN {X 0,Y 190.431,Z 376.957,A -85,B 0,C 180,E1 -22978.22,E2 -22978.22} C_VEL
LIN {X 0,Y 191.824,Z 364.506,A -85,B 0,C 180,E1 -22979.155,E2 -22979.155} C_VEL
LIN {X 0,Y 192.881,Z 348.984,A -85,B 0,C 180,E1 -22979.81,E2 -22979.81} C_VEL
LIN {X 0,Y 195.125,Z 303.124,A -85,B 0,C 180,E1 -22981.373,E2 -22981.373} C_VEL
LIN {X 0,Y 189.744,Z 289.533,A -85,B 0,C 180,E1 -22983.135,E2 -22983.135} C_VEL
LIN {X 0,Y 182.902,Z 276.963,A -85,B 0,C 180,E1 -22985.359,E2 -22985.359} C_VEL
LIN {X 0,Y 176.27,Z 266.42,A -85,B 0,C 180,E1 -22987.668,E2 -22987.668} C_VEL
LIN {X 0,Y 173.806,Z 262.665,A -85,B 0,C 180,E1 -22988.584,E2 -22988.584} C_VEL
LIN {X 0,Y 172.036,Z 260.435,A -85,B 0,C 180,E1 -22989.24,E2 -22989.24} C_VEL
LIN {X 0,Y 171.342,Z 258.14,A -85,B 0,C 180,E1 -22989.624,E2 -22989.624} C_VEL
LIN {X 0,Y 171.323,Z 258.144,A -85,B 0,C 180,E1 -22994.216,E2 -22994.216} C_VEL
LIN {X 0,Y 171.337,Z 258.143,A -85,B 0,C 180,E1 -22998.981,E2 -22998.981} C_VEL
LIN {X 0,Y 171.388,Z 258.132,A -85,B 0,C 180,E1 -23002.041,E2 -23002.041} C_VEL
LIN {X 0,Y 171.399,Z 258.125,A -85,B 0,C 180,E1 -23005.092,E2 -23005.092} C_VEL
LIN {X 0,Y 171.449,Z 258.119,A -85,B 0,C 180,E1 -23010.534,E2 -23010.534} C_VEL
LIN {X 0,Y 171.458,Z 258.098,A -85,B 0,C 180,E1 -23015.801,E2 -23015.801} C_VEL
LIN {X 0,Y 171.58,Z 258.097,A -85,B 0,C 180,E1 -23020.871,E2 -23020.871} C_VEL
LIN {X 0,Y 171.577,Z 258.092,A -85,B 0,C 180,E1 -23025.772,E2 -23025.772} C_VEL
LIN {X 0,Y 171.844,Z 258.042,A -85,B 0,C 180,E1 -23030.584,E2 -23030.584} C_VEL
LIN {X 0,Y 171.808,Z 258.079,A -85,B 0,C 180,E1 -23035.307,E2 -23035.307} C_VEL
LIN {X 0,Y 172.331,Z 258.015,A -85,B 0,C 180,E1 -23040,E2 -23040} C_VEL
LIN {X 0,Y 171.822,Z 258.072,A -85,B 0,C 180,E1 -23044.692,E2 -23044.692} C_VEL
LIN {X 0,Y 171.904,Z 258.062,A -85,B 0,C 180,E1 -23049.412,E2 -23049.412} C_VEL
LIN {X 0,Y 171.563,Z 258.112,A -85,B 0,C 180,E1 -23054.228,E2 -23054.228} C_VEL
LIN {X 0,Y 171.515,Z 258.107,A -85,B 0,C 180,E1 -23059.533,E2 -23059.533} C_VEL
LIN {X 0,Y 171.444,Z 258.118,A -85,B 0,C 180,E1 -23065.598,E2 -23065.598} C_VEL
LIN {X 0,Y 171.417,Z 258.123,A -85,B 0,C 180,E1 -23070.573,E2 -23070.573} C_VEL
LIN {X 0,Y 171.392,Z 258.128,A -85,B 0,C 180,E1 -23075.035,E2 -23075.035} C_VEL
LIN {X 0,Y 171.345,Z 258.136,A -85,B 0,C 180,E1 -23078.802,E2 -23078.802} C_VEL
LIN {X 0,Y 171.387,Z 258.184,A -85,B 0,C 180,E1 -23083.319,E2 -23083.319} C_VEL
LIN {X 0,Y 171.748,Z 259.711,A -85,B 0,C 180,E1 -23084.278,E2 -23084.278} C_VEL
LIN {X 0,Y 174.272,Z 264.092,A -85,B 0,C 180,E1 -23085.277,E2 -23085.277} C_VEL
LIN {X 0,Y 180.769,Z 275.824,A -85,B 0,C 180,E1 -23087.684,E2 -23087.684} C_VEL
LIN {X 0,Y 186.726,Z 288.335,A -85,B 0,C 180,E1 -23089.764,E2 -23089.764} C_VEL
LIN {X 0,Y 192.926,Z 304.292,A -85,B 0,C 180,E1 -23091.87,E2 -23091.87} C_VEL
LIN {X 0,Y 194.445,Z 319.625,A -85,B 0,C 180,E1 -23092.86,E2 -23092.86} C_VEL
LIN {X 0,Y 191.965,Z 368.158,A -85,B 0,C 180,E1 -23094.546,E2 -23094.546} C_VEL
LIN {X 0,Y 190.56,Z 381.591,A -85,B 0,C 180,E1 -23095.376,E2 -23095.376} C_VEL
LIN {X 0,Y 189.634,Z 387.751,A -85,B 0,C 180,E1 -23095.889,E2 -23095.889} C_VEL
LIN {X 0,Y 188.286,Z 393.275,A -85,B 0,C 180,E1 -23096.359,E2 -23096.359} C_VEL
LIN {X 0,Y 184.143,Z 402.03,A -85,B 0,C 180,E1 -23096.996,E2 -23096.996} C_VEL
LIN {X 0,Y 179.566,Z 410.476,A -85,B 0,C 180,E1 -23097.833,E2 -23097.833} C_VEL
LIN {X 0,Y 177.575,Z 415.463,A -85,B 0,C 180,E1 -23098.621,E2 -23098.621} C_VEL
LIN {X 0,Y 174.363,Z 426.584,A -85,B 0,C 180,E1 -23101.074,E2 -23101.074} C_VEL
LIN {X 0,Y 171.343,Z 436.288,A -85,B 0,C 180,E1 -23103.837,E2 -23103.837} C_VEL
LIN {X 0,Y 168.851,Z 444.623,A -85,B 0,C 180,E1 -23106.873,E2 -23106.873} C_VEL
LIN {X 0,Y 166.359,Z 452.005,A -85,B 0,C 180,E1 -23110.247,E2 -23110.247} C_VEL
LIN {X 0,Y 164.295,Z 458.219,A -85,B 0,C 180,E1 -23113.856,E2 -23113.856} C_VEL
LIN {X 0,Y 162.961,Z 463.156,A -85,B 0,C 180,E1 -23117.547,E2 -23117.547} C_VEL
LIN {X 0,Y 162.172,Z 466.953,A -85,B 0,C 180,E1 -23121.276,E2 -23121.276} C_VEL
LIN {X 0,Y 161.848,Z 469.716,A -85,B 0,C 180,E1 -23125.018,E2 -23125.018} C_VEL
LIN {X 0,Y 161.817,Z 471.015,A -85,B 0,C 180,E1 -23127.511,E2 -23127.511} C_VEL
LIN {X 0,Y 161.911,Z 471.917,A -85,B 0,C 180,E1 -23130,E2 -23130} C_VEL
LIN {X 0,Y 161.797,Z 472.391,A -85,B 0,C 180,E1 -23132.49,E2 -23132.49} C_VEL
LIN {X 0,Y 161.85,Z 472.446,A -85,B 0,C 180,E1 -23134.982,E2 -23134.982} C_VEL
LIN {X 0,Y 162.441,Z 471.407,A -85,B 0,C 180,E1 -23139.966,E2 -23139.966} C_VEL
LIN {X 0,Y 163.133,Z 470.3,A -85,B 0,C 180,E1 -23142.439,E2 -23142.439} C_VEL
LIN {X 0,Y 165.213,Z 466.788,A -85,B 0,C 180,E1 -23147.324,E2 -23147.324} C_VEL
LIN {X 0,Y 167.706,Z 463.006,A -85,B 0,C 180,E1 -23150.868,E2 -23150.868} C_VEL
LIN {X 0,Y 170.754,Z 458.118,A -85,B 0,C 180,E1 -23154.305,E2 -23154.305} C_VEL
LIN {X 0,Y 174.137,Z 452.202,A -85,B 0,C 180,E1 -23157.524,E2 -23157.524} C_VEL
LIN {X 0,Y 178.331,Z 444.363,A -85,B 0,C 180,E1 -23160.819,E2 -23160.819} C_VEL
LIN {X 0,Y 182.333,Z 436.581,A -85,B 0,C 180,E1 -23163.317,E2 -23163.317} C_VEL
LIN {X 0,Y 187.034,Z 426.026,A -85,B 0,C 180,E1 -23165.953,E2 -23165.953} C_VEL
LIN {X 0,Y 191.25,Z 415.295,A -85,B 0,C 180,E1 -23167.99,E2 -23167.99} C_VEL
LIN {X 0,Y 194.708,Z 404.873,A -85,B 0,C 180,E1 -23169.507,E2 -23169.507} C_VEL
LIN {X 0,Y 197.739,Z 393.475,A -85,B 0,C 180,E1 -23170.774,E2 -23170.774} C_VEL
LIN {X 0,Y 200.354,Z 380.653,A -85,B 0,C 180,E1 -23171.796,E2 -23171.796} C_VEL
LIN {X 0,Y 202.109,Z 368.202,A -85,B 0,C 180,E1 -23172.449,E2 -23172.449} C_VEL
LIN {X 0,Y 204.718,Z 327.795,A -85,B 0,C 180,E1 -23173.771,E2 -23173.771} C_VEL
LIN {X 0,Y 199.161,Z 314.095,A -85,B 0,C 180,E1 -23176.203,E2 -23176.203} C_VEL
LIN {X 0,Y 193.953,Z 303.231,A -85,B 0,C 180,E1 -23178.617,E2 -23178.617} C_VEL
LIN {X 0,Y 187.816,Z 291.923,A -85,B 0,C 180,E1 -23181.731,E2 -23181.731} C_VEL
LIN {X 0,Y 183.812,Z 285.546,A -85,B 0,C 180,E1 -23183.953,E2 -23183.953} C_VEL
LIN {X 0,Y 181.291,Z 281.484,A -85,B 0,C 180,E1 -23185.478,E2 -23185.478} C_VEL
LIN {X 0,Y 177.826,Z 276.285,A -85,B 0,C 180,E1 -23187.734,E2 -23187.734} C_VEL
LIN {X 0,Y 173.988,Z 270.879,A -85,B 0,C 180,E1 -23190.52,E2 -23190.52} C_VEL
LIN {X 0,Y 173.11,Z 270.054,A -85,B 0,C 180,E1 -23191.177,E2 -23191.177} C_VEL
LIN {X 0,Y 170.592,Z 267.598,A -85,B 0,C 180,E1 -23193.205,E2 -23193.205} C_VEL
LIN {X 0,Y 169.085,Z 264.817,A -85,B 0,C 180,E1 -23194.672,E2 -23194.672} C_VEL
LIN {X 0,Y 166.298,Z 263.053,A -85,B 0,C 180,E1 -23197.317,E2 -23197.317} C_VEL
LIN {X 0,Y 164.838,Z 260.717,A -85,B 0,C 180,E1 -23199.079,E2 -23199.079} C_VEL
LIN {X 0,Y 164.437,Z 258.993,A -85,B 0,C 180,E1 -23199.843,E2 -23199.843} C_VEL
LIN {X 0,Y 164.492,Z 258.991,A -85,B 0,C 180,E1 -23205.146,E2 -23205.146} C_VEL
LIN {X 0,Y 164.803,Z 258.954,A -85,B 0,C 180,E1 -23210.179,E2 -23210.179} C_VEL
LIN {X 0,Y 164.85,Z 258.934,A -85,B 0,C 180,E1 -23212.652,E2 -23212.652} C_VEL
LIN {X 0,Y 165.046,Z 258.91,A -85,B 0,C 180,E1 -23217.56,E2 -23217.56} C_VEL
LIN {X 0,Y 165.294,Z 258.89,A -85,B 0,C 180,E1 -23220,E2 -23220} C_VEL
LIN {X 0,Y 164.754,Z 258.955,A -85,B 0,C 180,E1 -23224.894,E2 -23224.894} C_VEL
LIN {X 0,Y 164.824,Z 258.941,A -85,B 0,C 180,E1 -23227.35,E2 -23227.35} C_VEL
LIN {X 0,Y 164.703,Z 258.969,A -85,B 0,C 180,E1 -23231.06,E2 -23231.06} C_VEL
LIN {X 0,Y 164.52,Z 259.031,A -85,B 0,C 180,E1 -23234.772,E2 -23234.772} C_VEL
LIN {X 0,Y 165.096,Z 261.09,A -85,B 0,C 180,E1 -23235.668,E2 -23235.668} C_VEL
LIN {X 0,Y 166.948,Z 263.526,A -85,B 0,C 180,E1 -23237.771,E2 -23237.771} C_VEL
LIN {X 0,Y 169.391,Z 265.063,A -85,B 0,C 180,E1 -23240.028,E2 -23240.028} C_VEL
LIN {X 0,Y 170.818,Z 267.857,A -85,B 0,C 180,E1 -23241.417,E2 -23241.417} C_VEL
LIN {X 0,Y 173.557,Z 270.299,A -85,B 0,C 180,E1 -23243.571,E2 -23243.571} C_VEL
LIN {X 0,Y 176.437,Z 274.35,A -85,B 0,C 180,E1 -23245.729,E2 -23245.729} C_VEL
LIN {X 0,Y 178.033,Z 275.935,A -85,B 0,C 180,E1 -23246.781,E2 -23246.781} C_VEL
LIN {X 0,Y 180.763,Z 279.649,A -85,B 0,C 180,E1 -23248.542,E2 -23248.542} C_VEL
LIN {X 0,Y 185.535,Z 286.13,A -85,B 0,C 180,E1 -23251.311,E2 -23251.311} C_VEL
LIN {X 0,Y 190.429,Z 293.142,A -85,B 0,C 180,E1 -23253.853,E2 -23253.853} C_VEL
LIN {X 0,Y 197.235,Z 304.084,A -85,B 0,C 180,E1 -23257.028,E2 -23257.028} C_VEL
LIN {X 0,Y 202.818,Z 315.639,A -85,B 0,C 180,E1 -23259.468,E2 -23259.468} C_VEL
LIN {X 0,Y 205.161,Z 321.188,A -85,B 0,C 180,E1 -23260.456,E2 -23260.456} C_VEL
LIN {X 0,Y 202.523,Z 360.609,A -85,B 0,C 180,E1 -23261.73,E2 -23261.73} C_VEL
LIN {X 0,Y 200.743,Z 374.053,A -85,B 0,C 180,E1 -23262.506,E2 -23262.506} C_VEL
LIN {X 0,Y 198.262,Z 386.565,A -85,B 0,C 180,E1 -23263.575,E2 -23263.575} C_VEL
LIN {X 0,Y 195.086,Z 398.573,A -85,B 0,C 180,E1 -23265.009,E2 -23265.009} C_VEL
LIN {X 0,Y 191.202,Z 410.044,A -85,B 0,C 180,E1 -23266.796,E2 -23266.796} C_VEL
LIN {X 0,Y 187.254,Z 420.267,A -85,B 0,C 180,E1 -23268.909,E2 -23268.909} C_VEL
LIN {X 0,Y 182.99,Z 429.597,A -85,B 0,C 180,E1 -23271.383,E2 -23271.383} C_VEL
LIN {X 0,Y 178.389,Z 438.558,A -85,B 0,C 180,E1 -23274.471,E2 -23274.471} C_VEL
LIN {X 0,Y 174.27,Z 446.01,A -85,B 0,C 180,E1 -23277.876,E2 -23277.876} C_VEL
LIN {X 0,Y 170.407,Z 452.249,A -85,B 0,C 180,E1 -23281.687,E2 -23281.687} C_VEL
LIN {X 0,Y 167.594,Z 456.53,A -85,B 0,C 180,E1 -23285.207,E2 -23285.207} C_VEL
LIN {X 0,Y 165.001,Z 460.267,A -85,B 0,C 180,E1 -23289.565,E2 -23289.565} C_VEL
LIN {X 0,Y 163.653,Z 461.933,A -85,B 0,C 180,E1 -23292.506,E2 -23292.506} C_VEL
LIN {X 0,Y 162.215,Z 463.438,A -85,B 0,C 180,E1 -23297.489,E2 -23297.489} C_VEL
LIN {X 0,Y 161.898,Z 463.575,A -85,B 0,C 180,E1 -23300,E2 -23300} C_VEL
LIN {X 0,Y 161.793,Z 463.3,A -85,B 0,C 180,E1 -23302.512,E2 -23302.512} C_VEL
LIN {X 0,Y 161.874,Z 461.863,A -85,B 0,C 180,E1 -23306.952,E2 -23306.952} C_VEL
LIN {X 0,Y 162.134,Z 460.145,A -85,B 0,C 180,E1 -23310,E2 -23310} C_VEL
LIN {X 0,Y 162.841,Z 457.162,A -85,B 0,C 180,E1 -23313.712,E2 -23313.712} C_VEL
LIN {X 0,Y 163.931,Z 453.145,A -85,B 0,C 180,E1 -23317.389,E2 -23317.389} C_VEL
LIN {X 0,Y 165.922,Z 446.967,A -85,B 0,C 180,E1 -23321.607,E2 -23321.607} C_VEL
LIN {X 0,Y 168.226,Z 440.246,A -85,B 0,C 180,E1 -23325.136,E2 -23325.136} C_VEL
LIN {X 0,Y 171.129,Z 431.891,A -85,B 0,C 180,E1 -23328.559,E2 -23328.559} C_VEL
LIN {X 0,Y 174.192,Z 422.244,A -85,B 0,C 180,E1 -23331.626,E2 -23331.626} C_VEL
LIN {X 0,Y 177.094,Z 412.299,A -85,B 0,C 180,E1 -23334.109,E2 -23334.109} C_VEL
LIN {X 0,Y 179.691,Z 402.18,A -85,B 0,C 180,E1 -23336.104,E2 -23336.104} C_VEL
LIN {X 0,Y 182.22,Z 390.478,A -85,B 0,C 180,E1 -23337.881,E2 -23337.881} C_VEL
LIN {X 0,Y 184.252,Z 378.329,A -85,B 0,C 180,E1 -23339.256,E2 -23339.256} C_VEL
LIN {X 0,Y 185.814,Z 365.459,A -85,B 0,C 180,E1 -23340.274,E2 -23340.274} C_VEL
LIN {X 0,Y 186.864,Z 351.588,A -85,B 0,C 180,E1 -23340.909,E2 -23340.909} C_VEL
LIN {X 0,Y 189.261,Z 305.005,A -85,B 0,C 180,E1 -23342.529,E2 -23342.529} C_VEL
LIN {X 0,Y 184.415,Z 292.742,A -85,B 0,C 180,E1 -23344.217,E2 -23344.217} C_VEL
LIN {X 0,Y 177.919,Z 280.849,A -85,B 0,C 180,E1 -23346.459,E2 -23346.459} C_VEL
LIN {X 0,Y 171.674,Z 270.845,A -85,B 0,C 180,E1 -23348.772,E2 -23348.772} C_VEL
LIN {X 0,Y 169.287,Z 267.362,A -85,B 0,C 180,E1 -23349.705,E2 -23349.705} C_VEL
LIN {X 0,Y 166.87,Z 263.669,A -85,B 0,C 180,E1 -23350.702,E2 -23350.702} C_VEL
LIN {X 0,Y 165.012,Z 261.347,A -85,B 0,C 180,E1 -23351.469,E2 -23351.469} C_VEL
LIN {X 0,Y 164.283,Z 259.019,A -85,B 0,C 180,E1 -23351.873,E2 -23351.873} C_VEL
LIN {X 0,Y 164.293,Z 259.019,A -85,B 0,C 180,E1 -23356.808,E2 -23356.808} C_VEL
LIN {X 0,Y 164.297,Z 259.016,A -85,B 0,C 180,E1 -23360.351,E2 -23360.351} C_VEL
LIN {X 0,Y 164.331,Z 259.011,A -85,B 0,C 180,E1 -23364.348,E2 -23364.348} C_VEL
LIN {X 0,Y 164.39,Z 258.981,A -85,B 0,C 180,E1 -23369.134,E2 -23369.134} C_VEL
LIN {X 0,Y 164.417,Z 258.99,A -85,B 0,C 180,E1 -23374.694,E2 -23374.694} C_VEL
LIN {X 0,Y 164.486,Z 258.97,A -85,B 0,C 180,E1 -23380.051,E2 -23380.051} C_VEL
LIN {X 0,Y 164.525,Z 258.977,A -85,B 0,C 180,E1 -23385.149,E2 -23385.149} C_VEL
LIN {X 0,Y 164.765,Z 258.918,A -85,B 0,C 180,E1 -23390.176,E2 -23390.176} C_VEL
LIN {X 0,Y 164.824,Z 258.939,A -85,B 0,C 180,E1 -23392.65,E2 -23392.65} C_VEL
LIN {X 0,Y 165.045,Z 258.912,A -85,B 0,C 180,E1 -23397.559,E2 -23397.559} C_VEL
LIN {X 0,Y 165.294,Z 258.892,A -85,B 0,C 180,E1 -23400,E2 -23400} C_VEL
LIN {X 0,Y 164.772,Z 258.951,A -85,B 0,C 180,E1 -23404.893,E2 -23404.893} C_VEL
LIN {X 0,Y 164.861,Z 258.949,A -85,B 0,C 180,E1 -23407.347,E2 -23407.347} C_VEL
LIN {X 0,Y 164.748,Z 258.942,A -85,B 0,C 180,E1 -23411.141,E2 -23411.141} C_VEL
LIN {X 0,Y 164.453,Z 258.987,A -85,B 0,C 180,E1 -23417.406,E2 -23417.406} C_VEL
LIN {X 0,Y 164.449,Z 258.99,A -85,B 0,C 180,E1 -23419.992,E2 -23419.992} C_VEL
LIN {X 0,Y 164.37,Z 259.001,A -85,B 0,C 180,E1 -23426.117,E2 -23426.117} C_VEL
LIN {X 0,Y 164.357,Z 259.004,A -85,B 0,C 180,E1 -23431.217,E2 -23431.217} C_VEL
LIN {X 0,Y 164.28,Z 259.022,A -85,B 0,C 180,E1 -23436.793,E2 -23436.793} C_VEL
LIN {X 0,Y 164.309,Z 259.214,A -85,B 0,C 180,E1 -23441.784,E2 -23441.784} C_VEL
LIN {X 0,Y 165.353,Z 261.95,A -85,B 0,C 180,E1 -23442.33,E2 -23442.33} C_VEL
LIN {X 0,Y 167.755,Z 265.053,A -85,B 0,C 180,E1 -23443.316,E2 -23443.316} C_VEL
LIN {X 0,Y 175.274,Z 278.412,A -85,B 0,C 180,E1 -23446.332,E2 -23446.332} C_VEL
LIN {X 0,Y 181.442,Z 291.546,A -85,B 0,C 180,E1 -23448.642,E2 -23448.642} C_VEL
LIN {X 0,Y 187.129,Z 306.321,A -85,B 0,C 180,E1 -23450.703,E2 -23450.703} C_VEL
LIN {X 0,Y 187.614,Z 309.089,A -85,B 0,C 180,E1 -23450.941,E2 -23450.941} C_VEL
LIN {X 0,Y 188.594,Z 320.055,A -85,B 0,C 180,E1 -23451.662,E2 -23451.662} C_VEL
LIN {X 0,Y 185.992,Z 368.511,A -85,B 0,C 180,E1 -23453.393,E2 -23453.393} C_VEL
LIN {X 0,Y 184.528,Z 381.755,A -85,B 0,C 180,E1 -23454.24,E2 -23454.24} C_VEL
LIN {X 0,Y 182.537,Z 393.906,A -85,B 0,C 180,E1 -23455.396,E2 -23455.396} C_VEL
LIN {X 0,Y 180.107,Z 405.346,A -85,B 0,C 180,E1 -23456.887,E2 -23456.887} C_VEL
LIN {X 0,Y 177.575,Z 415.463,A -85,B 0,C 180,E1 -23458.621,E2 -23458.621} C_VEL
LIN {X 0,Y 175.558,Z 420.324,A -85,B 0,C 180,E1 -23459.501,E2 -23459.501} C_VEL
LIN {X 0,Y 168.631,Z 430.75,A -85,B 0,C 180,E1 -23461.508,E2 -23461.508} C_VEL
LIN {X 0,Y 165.064,Z 436.346,A -85,B 0,C 180,E1 -23462.981,E2 -23462.981} C_VEL
LIN {X 0,Y 163.884,Z 439.019,A -85,B 0,C 180,E1 -23463.881,E2 -23463.881} C_VEL
LIN {X 0,Y 161.482,Z 446.557,A -85,B 0,C 180,E1 -23466.94,E2 -23466.94} C_VEL
LIN {X 0,Y 158.859,Z 453.844,A -85,B 0,C 180,E1 -23470.622,E2 -23470.622} C_VEL
LIN {X 0,Y 156.845,Z 459.663,A -85,B 0,C 180,E1 -23474.404,E2 -23474.404} C_VEL
LIN {X 0,Y 155.653,Z 464.245,A -85,B 0,C 180,E1 -23478.277,E2 -23478.277} C_VEL
LIN {X 0,Y 154.95,Z 467.719,A -85,B 0,C 180,E1 -23482.18,E2 -23482.18} C_VEL
LIN {X 0,Y 154.751,Z 469.449,A -85,B 0,C 180,E1 -23484.789,E2 -23484.789} C_VEL
LIN {X 0,Y 154.742,Z 470.892,A -85,B 0,C 180,E1 -23487.69,E2 -23487.69} C_VEL
LIN {X 0,Y 154.81,Z 471.682,A -85,B 0,C 180,E1 -23490,E2 -23490} C_VEL
LIN {X 0,Y 154.698,Z 472.184,A -85,B 0,C 180,E1 -23492.604,E2 -23492.604} C_VEL
LIN {X 0,Y 154.755,Z 472.256,A -85,B 0,C 180,E1 -23495.211,E2 -23495.211} C_VEL
LIN {X 0,Y 155.441,Z 471.249,A -85,B 0,C 180,E1 -23500.42,E2 -23500.42} C_VEL
LIN {X 0,Y 156.181,Z 470.166,A -85,B 0,C 180,E1 -23503.003,E2 -23503.003} C_VEL
LIN {X 0,Y 157.15,Z 468.638,A -85,B 0,C 180,E1 -23505.565,E2 -23505.565} C_VEL
LIN {X 0,Y 159.257,Z 465.576,A -85,B 0,C 180,E1 -23509.328,E2 -23509.328} C_VEL
LIN {X 0,Y 162.04,Z 461.476,A -85,B 0,C 180,E1 -23512.976,E2 -23512.976} C_VEL
LIN {X 0,Y 165.512,Z 456.223,A -85,B 0,C 180,E1 -23516.478,E2 -23516.478} C_VEL
LIN {X 0,Y 169.326,Z 449.648,A -85,B 0,C 180,E1 -23519.872,E2 -23519.872} C_VEL
LIN {X 0,Y 173.874,Z 441.496,A -85,B 0,C 180,E1 -23523.071,E2 -23523.071} C_VEL
LIN {X 0,Y 178.175,Z 433.174,A -85,B 0,C 180,E1 -23525.578,E2 -23525.578} C_VEL
LIN {X 0,Y 182.732,Z 422.963,A -85,B 0,C 180,E1 -23527.979,E2 -23527.979} C_VEL
LIN {X 0,Y 187.233,Z 411.435,A -85,B 0,C 180,E1 -23530.002,E2 -23530.002} C_VEL
LIN {X 0,Y 190.836,Z 400.086,A -85,B 0,C 180,E1 -23531.521,E2 -23531.521} C_VEL
LIN {X 0,Y 193.758,Z 388.429,A -85,B 0,C 180,E1 -23532.675,E2 -23532.675} C_VEL
LIN {X 0,Y 196.202,Z 375.013,A -85,B 0,C 180,E1 -23533.595,E2 -23533.595} C_VEL
LIN {X 0,Y 197.696,Z 362.256,A -85,B 0,C 180,E1 -23534.122,E2 -23534.122} C_VEL
LIN {X 0,Y 199.728,Z 330.083,A -85,B 0,C 180,E1 -23535.172,E2 -23535.172} C_VEL
LIN {X 0,Y 194.596,Z 317.213,A -85,B 0,C 180,E1 -23537.585,E2 -23537.585} C_VEL
LIN {X 0,Y 188.991,Z 305.397,A -85,B 0,C 180,E1 -23540.395,E2 -23540.395} C_VEL
LIN {X 0,Y 183.704,Z 295.862,A -85,B 0,C 180,E1 -23543.291,E2 -23543.291} C_VEL
LIN {X 0,Y 180.549,Z 290.572,A -85,B 0,C 180,E1 -23545.186,E2 -23545.186} C_VEL
LIN {X 0,Y 178.352,Z 286.968,A -85,B 0,C 180,E1 -23546.603,E2 -23546.603} C_VEL
LIN {X 0,Y 175.198,Z 282.093,A -85,B 0,C 180,E1 -23548.79,E2 -23548.79} C_VEL
LIN {X 0,Y 171.602,Z 276.891,A -85,B 0,C 180,E1 -23551.569,E2 -23551.569} C_VEL
LIN {X 0,Y 168.799,Z 274.208,A -85,B 0,C 180,E1 -23553.899,E2 -23553.899} C_VEL
LIN {X 0,Y 167.227,Z 271.509,A -85,B 0,C 180,E1 -23555.48,E2 -23555.48} C_VEL
LIN {X 0,Y 164.537,Z 269.47,A -85,B 0,C 180,E1 -23558.218,E2 -23558.218} C_VEL
LIN {X 0,Y 162.929,Z 266.476,A -85,B 0,C 180,E1 -23560.365,E2 -23560.365} C_VEL
LIN {X 0,Y 162.741,Z 265.892,A -85,B 0,C 180,E1 -23560.672,E2 -23560.672} C_VEL
LIN {X 0,Y 159.747,Z 264.263,A -85,B 0,C 180,E1 -23565.105,E2 -23565.105} C_VEL
LIN {X 0,Y 158.258,Z 261.901,A -85,B 0,C 180,E1 -23568.611,E2 -23568.611} C_VEL
LIN {X 0,Y 157.756,Z 259.831,A -85,B 0,C 180,E1 -23570.868,E2 -23570.868} C_VEL
LIN {X 0,Y 157.97,Z 259.791,A -85,B 0,C 180,E1 -23577.45,E2 -23577.45} C_VEL
LIN {X 0,Y 158.256,Z 259.766,A -85,B 0,C 180,E1 -23580,E2 -23580} C_VEL
LIN {X 0,Y 157.803,Z 259.862,A -85,B 0,C 180,E1 -23583.911,E2 -23583.911} C_VEL
LIN {X 0,Y 158.192,Z 261.643,A -85,B 0,C 180,E1 -23585.577,E2 -23585.577} C_VEL
LIN {X 0,Y 160.714,Z 264.839,A -85,B 0,C 180,E1 -23590.938,E2 -23590.938} C_VEL
LIN {X 0,Y 162.893,Z 266.11,A -85,B 0,C 180,E1 -23593.966,E2 -23593.966} C_VEL
LIN {X 0,Y 164.123,Z 268.704,A -85,B 0,C 180,E1 -23595.683,E2 -23595.683} C_VEL
LIN {X 0,Y 166.274,Z 270.897,A -85,B 0,C 180,E1 -23598.039,E2 -23598.039} C_VEL
LIN {X 0,Y 167.488,Z 271.672,A -85,B 0,C 180,E1 -23599.186,E2 -23599.186} C_VEL
LIN {X 0,Y 169.424,Z 274.937,A -85,B 0,C 180,E1 -23601.086,E2 -23601.086} C_VEL
LIN {X 0,Y 171.931,Z 277.372,A -85,B 0,C 180,E1 -23603.129,E2 -23603.129} C_VEL
LIN {X 0,Y 174.538,Z 280.957,A -85,B 0,C 180,E1 -23605.139,E2 -23605.139} C_VEL
LIN {X 0,Y 175.772,Z 282.324,A -85,B 0,C 180,E1 -23605.997,E2 -23605.997} C_VEL
LIN {X 0,Y 178.711,Z 286.224,A -85,B 0,C 180,E1 -23607.959,E2 -23607.959} C_VEL
LIN {X 0,Y 184.846,Z 294.963,A -85,B 0,C 180,E1 -23611.595,E2 -23611.595} C_VEL
LIN {X 0,Y 191.32,Z 305.235,A -85,B 0,C 180,E1 -23614.938,E2 -23614.938} C_VEL
LIN {X 0,Y 194.795,Z 311.507,A -85,B 0,C 180,E1 -23616.589,E2 -23616.589} C_VEL
LIN {X 0,Y 200.213,Z 323.56,A -85,B 0,C 180,E1 -23619.065,E2 -23619.065} C_VEL
LIN {X 0,Y 197.497,Z 361.468,A -85,B 0,C 180,E1 -23620.304,E2 -23620.304} C_VEL
LIN {X 0,Y 195.728,Z 374.266,A -85,B 0,C 180,E1 -23621.058,E2 -23621.058} C_VEL
LIN {X 0,Y 193.124,Z 386.863,A -85,B 0,C 180,E1 -23622.143,E2 -23622.143} C_VEL
LIN {X 0,Y 190.076,Z 398.047,A -85,B 0,C 180,E1 -23623.479,E2 -23623.479} C_VEL
LIN {X 0,Y 186.029,Z 409.652,A -85,B 0,C 180,E1 -23625.28,E2 -23625.28} C_VEL
LIN {X 0,Y 182.001,Z 419.708,A -85,B 0,C 180,E1 -23627.354,E2 -23627.354} C_VEL
LIN {X 0,Y 177.452,Z 429.424,A -85,B 0,C 180,E1 -23629.94,E2 -23629.94} C_VEL
LIN {X 0,Y 173.327,Z 437.085,A -85,B 0,C 180,E1 -23632.539,E2 -23632.539} C_VEL
LIN {X 0,Y 169.046,Z 444.576,A -85,B 0,C 180,E1 -23635.859,E2 -23635.859} C_VEL
LIN {X 0,Y 165.266,Z 450.565,A -85,B 0,C 180,E1 -23639.316,E2 -23639.316} C_VEL
LIN {X 0,Y 162.012,Z 455.28,A -85,B 0,C 180,E1 -23642.904,E2 -23642.904} C_VEL
LIN {X 0,Y 159.392,Z 458.867,A -85,B 0,C 180,E1 -23646.619,E2 -23646.619} C_VEL
LIN {X 0,Y 158.019,Z 460.703,A -85,B 0,C 180,E1 -23649.157,E2 -23649.157} C_VEL
LIN {X 0,Y 155.889,Z 463.033,A -85,B 0,C 180,E1 -23654.306,E2 -23654.306} C_VEL
LIN {X 0,Y 155.213,Z 463.609,A -85,B 0,C 180,E1 -23656.915,E2 -23656.915} C_VEL
LIN {X 0,Y 154.851,Z 463.782,A -85,B 0,C 180,E1 -23659.54,E2 -23659.54} C_VEL
LIN {X 0,Y 154.706,Z 463.525,A -85,B 0,C 180,E1 -23662.167,E2 -23662.167} C_VEL
LIN {X 0,Y 154.726,Z 462.887,A -85,B 0,C 180,E1 -23664.788,E2 -23664.788} C_VEL
LIN {X 0,Y 154.817,Z 461.869,A -85,B 0,C 180,E1 -23667.398,E2 -23667.398} C_VEL
LIN {X 0,Y 155.034,Z 460.443,A -85,B 0,C 180,E1 -23670,E2 -23670} C_VEL
LIN {X 0,Y 155.771,Z 457.493,A -85,B 0,C 180,E1 -23673.88,E2 -23673.88} C_VEL
LIN {X 0,Y 156.927,Z 453.515,A -85,B 0,C 180,E1 -23677.721,E2 -23677.721} C_VEL
LIN {X 0,Y 159.006,Z 447.39,A -85,B 0,C 180,E1 -23682.119,E2 -23682.119} C_VEL
LIN {X 0,Y 161.423,Z 440.719,A -85,B 0,C 180,E1 -23685.79,E2 -23685.79} C_VEL
LIN {X 0,Y 164.457,Z 432.439,A -85,B 0,C 180,E1 -23689.341,E2 -23689.341} C_VEL
LIN {X 0,Y 167.628,Z 422.88,A -85,B 0,C 180,E1 -23692.519,E2 -23692.519} C_VEL
LIN {X 0,Y 170.827,Z 412.523,A -85,B 0,C 180,E1 -23695.193,E2 -23695.193} C_VEL
LIN {X 0,Y 173.747,Z 401.572,A -85,B 0,C 180,E1 -23697.394,E2 -23697.394} C_VEL
LIN {X 0,Y 176.4,Z 389.591,A -85,B 0,C 180,E1 -23699.213,E2 -23699.213} C_VEL
LIN {X 0,Y 178.537,Z 377.107,A -85,B 0,C 180,E1 -23700.616,E2 -23700.616} C_VEL
LIN {X 0,Y 180.025,Z 364.784,A -85,B 0,C 180,E1 -23701.579,E2 -23701.579} C_VEL
LIN {X 0,Y 181.133,Z 349.767,A -85,B 0,C 180,E1 -23702.243,E2 -23702.243} C_VEL
LIN {X 0,Y 183.478,Z 306.896,A -85,B 0,C 180,E1 -23703.758,E2 -23703.758} C_VEL
LIN {X 0,Y 179.407,Z 296.536,A -85,B 0,C 180,E1 -23705.27,E2 -23705.27} C_VEL
LIN {X 0,Y 173.373,Z 285.329,A -85,B 0,C 180,E1 -23707.483,E2 -23707.483} C_VEL
LIN {X 0,Y 167.073,Z 275.093,A -85,B 0,C 180,E1 -23709.969,E2 -23709.969} C_VEL
LIN {X 0,Y 162.685,Z 268.663,A -85,B 0,C 180,E1 -23711.839,E2 -23711.839} C_VEL
LIN {X 0,Y 160.509,Z 265.292,A -85,B 0,C 180,E1 -23712.84,E2 -23712.84} C_VEL
LIN {X 0,Y 157.984,Z 262.382,A -85,B 0,C 180,E1 -23713.994,E2 -23713.994} C_VEL
LIN {X 0,Y 157.179,Z 259.905,A -85,B 0,C 180,E1 -23714.519,E2 -23714.519} C_VEL
LIN {X 0,Y 157.206,Z 259.903,A -85,B 0,C 180,E1 -23719.464,E2 -23719.464} C_VEL
LIN {X 0,Y 157.28,Z 259.888,A -85,B 0,C 180,E1 -23724.486,E2 -23724.486} C_VEL
LIN {X 0,Y 157.293,Z 259.858,A -85,B 0,C 180,E1 -23728.096,E2 -23728.096} C_VEL
LIN {X 0,Y 157.323,Z 259.885,A -85,B 0,C 180,E1 -23733.466,E2 -23733.466} C_VEL
LIN {X 0,Y 157.395,Z 259.846,A -85,B 0,C 180,E1 -23739.668,E2 -23739.668} C_VEL
LIN {X 0,Y 157.455,Z 259.862,A -85,B 0,C 180,E1 -23744.466,E2 -23744.466} C_VEL
LIN {X 0,Y 157.687,Z 259.794,A -85,B 0,C 180,E1 -23749.73,E2 -23749.73} C_VEL
LIN {X 0,Y 157.762,Z 259.814,A -85,B 0,C 180,E1 -23752.319,E2 -23752.319} C_VEL
LIN {X 0,Y 158.256,Z 259.768,A -85,B 0,C 180,E1 -23760,E2 -23760} C_VEL
LIN {X 0,Y 157.821,Z 259.826,A -85,B 0,C 180,E1 -23767.677,E2 -23767.677} C_VEL
LIN {X 0,Y 157.677,Z 259.823,A -85,B 0,C 180,E1 -23771.308,E2 -23771.308} C_VEL
LIN {X 0,Y 157.424,Z 259.874,A -85,B 0,C 180,E1 -23775.537,E2 -23775.537} C_VEL
LIN {X 0,Y 157.357,Z 259.88,A -85,B 0,C 180,E1 -23780.934,E2 -23780.934} C_VEL
LIN {X 0,Y 157.31,Z 259.884,A -85,B 0,C 180,E1 -23786.681,E2 -23786.681} C_VEL
LIN {X 0,Y 157.268,Z 259.894,A -85,B 0,C 180,E1 -23792.429,E2 -23792.429} C_VEL
LIN {X 0,Y 157.259,Z 259.893,A -85,B 0,C 180,E1 -23796.445,E2 -23796.445} C_VEL
LIN {X 0,Y 157.228,Z 259.894,A -85,B 0,C 180,E1 -23799.136,E2 -23799.136} C_VEL
LIN {X 0,Y 158.307,Z 262.8,A -85,B 0,C 180,E1 -23799.807,E2 -23799.807} C_VEL
LIN {X 0,Y 160.557,Z 265.351,A -85,B 0,C 180,E1 -23800.829,E2 -23800.829} C_VEL
LIN {X 0,Y 162.702,Z 268.679,A -85,B 0,C 180,E1 -23801.815,E2 -23801.815} C_VEL
LIN {X 0,Y 163.937,Z 270.552,A -85,B 0,C 180,E1 -23802.361,E2 -23802.361} C_VEL
LIN {X 0,Y 169.312,Z 280.158,A -85,B 0,C 180,E1 -23804.673,E2 -23804.673} C_VEL
LIN {X 0,Y 174.334,Z 290.379,A -85,B 0,C 180,E1 -23806.703,E2 -23806.703} C_VEL
LIN {X 0,Y 179.205,Z 302.214,A -85,B 0,C 180,E1 -23808.61,E2 -23808.61} C_VEL
LIN {X 0,Y 181.884,Z 309.816,A -85,B 0,C 180,E1 -23809.648,E2 -23809.648} C_VEL
LIN {X 0,Y 182.81,Z 320.229,A -85,B 0,C 180,E1 -23810.372,E2 -23810.372} C_VEL
LIN {X 0,Y 180.101,Z 368.991,A -85,B 0,C 180,E1 -23812.177,E2 -23812.177} C_VEL
LIN {X 0,Y 178.569,Z 381.945,A -85,B 0,C 180,E1 -23813.033,E2 -23813.033} C_VEL
LIN {X 0,Y 176.502,Z 393.965,A -85,B 0,C 180,E1 -23814.209,E2 -23814.209} C_VEL
LIN {X 0,Y 173.772,Z 406.133,A -85,B 0,C 180,E1 -23815.864,E2 -23815.864} C_VEL
LIN {X 0,Y 170.697,Z 417.708,A -85,B 0,C 180,E1 -23817.988,E2 -23817.988} C_VEL
LIN {X 0,Y 167.43,Z 428.121,A -85,B 0,C 180,E1 -23820.448,E2 -23820.448} C_VEL
LIN {X 0,Y 164.401,Z 437.48,A -85,B 0,C 180,E1 -23823.329,E2 -23823.329} C_VEL
LIN {X 0,Y 163.884,Z 439.019,A -85,B 0,C 180,E1 -23823.881,E2 -23823.881} C_VEL
LIN {X 0,Y 161.951,Z 442.94,A -85,B 0,C 180,E1 -23825.289,E2 -23825.289} C_VEL
LIN {X 0,Y 157.175,Z 448.814,A -85,B 0,C 180,E1 -23827.596,E2 -23827.596} C_VEL
LIN {X 0,Y 152.507,Z 454.116,A -85,B 0,C 180,E1 -23830.196,E2 -23830.196} C_VEL
LIN {X 0,Y 150.794,Z 456.997,A -85,B 0,C 180,E1 -23832.024,E2 -23832.024} C_VEL
LIN {X 0,Y 149.042,Z 462.485,A -85,B 0,C 180,E1 -23836.363,E2 -23836.363} C_VEL
LIN {X 0,Y 148.112,Z 466.354,A -85,B 0,C 180,E1 -23840.44,E2 -23840.44} C_VEL
LIN {X 0,Y 147.683,Z 469.182,A -85,B 0,C 180,E1 -23844.539,E2 -23844.539} C_VEL
LIN {X 0,Y 147.659,Z 470.907,A -85,B 0,C 180,E1 -23848.224,E2 -23848.224} C_VEL
LIN {X 0,Y 147.63,Z 471.745,A -85,B 0,C 180,E1 -23851.363,E2 -23851.363} C_VEL
LIN {X 0,Y 147.687,Z 472.067,A -85,B 0,C 180,E1 -23855.461,E2 -23855.461} C_VEL
LIN {X 0,Y 148.43,Z 471.09,A -85,B 0,C 180,E1 -23860.918,E2 -23860.918} C_VEL
LIN {X 0,Y 149.229,Z 470.028,A -85,B 0,C 180,E1 -23863.62,E2 -23863.62} C_VEL
LIN {X 0,Y 150.282,Z 468.527,A -85,B 0,C 180,E1 -23866.296,E2 -23866.296} C_VEL
LIN {X 0,Y 152.568,Z 465.499,A -85,B 0,C 180,E1 -23870.211,E2 -23870.211} C_VEL
LIN {X 0,Y 155.504,Z 461.435,A -85,B 0,C 180,E1 -23874.001,E2 -23874.001} C_VEL
LIN {X 0,Y 159.733,Z 455.305,A -85,B 0,C 180,E1 -23878.163,E2 -23878.163} C_VEL
LIN {X 0,Y 163.946,Z 448.458,A -85,B 0,C 180,E1 -23881.677,E2 -23881.677} C_VEL
LIN {X 0,Y 168.846,Z 440.085,A -85,B 0,C 180,E1 -23884.913,E2 -23884.913} C_VEL
LIN {X 0,Y 173.386,Z 431.47,A -85,B 0,C 180,E1 -23887.446,E2 -23887.446} C_VEL
LIN {X 0,Y 178.219,Z 420.878,A -85,B 0,C 180,E1 -23889.852,E2 -23889.852} C_VEL
LIN {X 0,Y 182.398,Z 410.367,A -85,B 0,C 180,E1 -23891.657,E2 -23891.657} C_VEL
LIN {X 0,Y 186.172,Z 398.725,A -85,B 0,C 180,E1 -23893.174,E2 -23893.174} C_VEL
LIN {X 0,Y 189.175,Z 386.648,A -85,B 0,C 180,E1 -23894.339,E2 -23894.339} C_VEL
LIN {X 0,Y 191.561,Z 373.716,A -85,B 0,C 180,E1 -23895.187,E2 -23895.187} C_VEL
LIN {X 0,Y 192.999,Z 360.899,A -85,B 0,C 180,E1 -23895.7,E2 -23895.7} C_VEL
LIN {X 0,Y 194.848,Z 332.414,A -85,B 0,C 180,E1 -23896.647,E2 -23896.647} C_VEL
LIN {X 0,Y 190.089,Z 320.249,A -85,B 0,C 180,E1 -23899.062,E2 -23899.062} C_VEL
LIN {X 0,Y 184.859,Z 309.159,A -85,B 0,C 180,E1 -23901.882,E2 -23901.882} C_VEL
LIN {X 0,Y 180.057,Z 300.197,A -85,B 0,C 180,E1 -23904.73,E2 -23904.73} C_VEL
LIN {X 0,Y 175.703,Z 292.767,A -85,B 0,C 180,E1 -23907.614,E2 -23907.614} C_VEL
LIN {X 0,Y 172.537,Z 287.757,A -85,B 0,C 180,E1 -23909.951,E2 -23909.951} C_VEL
LIN {X 0,Y 169.496,Z 283.292,A -85,B 0,C 180,E1 -23912.446,E2 -23912.446} C_VEL
LIN {X 0,Y 166.766,Z 280.387,A -85,B 0,C 180,E1 -23914.874,E2 -23914.874} C_VEL
LIN {X 0,Y 165.436,Z 278.151,A -85,B 0,C 180,E1 -23916.281,E2 -23916.281} C_VEL
LIN {X 0,Y 162.868,Z 275.903,A -85,B 0,C 180,E1 -23919.083,E2 -23919.083} C_VEL
LIN {X 0,Y 161.28,Z 272.813,A -85,B 0,C 180,E1 -23921.367,E2 -23921.367} C_VEL
LIN {X 0,Y 158.299,Z 270.81,A -85,B 0,C 180,E1 -23926.203,E2 -23926.203} C_VEL
LIN {X 0,Y 157.041,Z 268.306,A -85,B 0,C 180,E1 -23929.688,E2 -23929.688} C_VEL
LIN {X 0,Y 156.701,Z 266.848,A -85,B 0,C 180,E1 -23931.293,E2 -23931.293} C_VEL
LIN {X 0,Y 156.283,Z 266.643,A -85,B 0,C 180,E1 -23941.289,E2 -23941.289} C_VEL
LIN {X 0,Y 156.756,Z 266.968,A -85,B 0,C 180,E1 -23943.374,E2 -23943.374} C_VEL
LIN {X 0,Y 157.408,Z 269.111,A -85,B 0,C 180,E1 -23945.927,E2 -23945.927} C_VEL
LIN {X 0,Y 160.304,Z 272.267,A -85,B 0,C 180,E1 -23951.69,E2 -23951.69} C_VEL
LIN {X 0,Y 161.391,Z 272.935,A -85,B 0,C 180,E1 -23953.216,E2 -23953.216} C_VEL
LIN {X 0,Y 163.109,Z 276.074,A -85,B 0,C 180,E1 -23955.623,E2 -23955.623} C_VEL
LIN {X 0,Y 165.757,Z 278.45,A -85,B 0,C 180,E1 -23958.466,E2 -23958.466} C_VEL
LIN {X 0,Y 167.909,Z 281.781,A -85,B 0,C 180,E1 -23960.626,E2 -23960.626} C_VEL
LIN {X 0,Y 169.912,Z 283.85,A -85,B 0,C 180,E1 -23962.335,E2 -23962.335} C_VEL
LIN {X 0,Y 172.737,Z 287.639,A -85,B 0,C 180,E1 -23964.593,E2 -23964.593} C_VEL
LIN {X 0,Y 177.059,Z 293.648,A -85,B 0,C 180,E1 -23967.64,E2 -23967.64} C_VEL
LIN {X 0,Y 181.745,Z 300.361,A -85,B 0,C 180,E1 -23970.529,E2 -23970.529} C_VEL
LIN {X 0,Y 187.931,Z 310.491,A -85,B 0,C 180,E1 -23973.92,E2 -23973.92} C_VEL
LIN {X 0,Y 191.129,Z 316.44,A -85,B 0,C 180,E1 -23975.532,E2 -23975.532} C_VEL
LIN {X 0,Y 195.314,Z 325.983,A -85,B 0,C 180,E1 -23977.582,E2 -23977.582} C_VEL
LIN {X 0,Y 192.685,Z 361.722,A -85,B 0,C 180,E1 -23978.78,E2 -23978.78} C_VEL
LIN {X 0,Y 190.824,Z 374.615,A -85,B 0,C 180,E1 -23979.545,E2 -23979.545} C_VEL
LIN {X 0,Y 188.125,Z 387.165,A -85,B 0,C 180,E1 -23980.638,E2 -23980.638} C_VEL
LIN {X 0,Y 184.7,Z 399.119,A -85,B 0,C 180,E1 -23982.098,E2 -23982.098} C_VEL
LIN {X 0,Y 180.494,Z 410.561,A -85,B 0,C 180,E1 -23983.917,E2 -23983.917} C_VEL
LIN {X 0,Y 176.409,Z 420.274,A -85,B 0,C 180,E1 -23985.975,E2 -23985.975} C_VEL
LIN {X 0,Y 172.043,Z 429.251,A -85,B 0,C 180,E1 -23988.408,E2 -23988.408} C_VEL
LIN {X 0,Y 167.66,Z 436.973,A -85,B 0,C 180,E1 -23991.04,E2 -23991.04} C_VEL
LIN {X 0,Y 163.112,Z 444.517,A -85,B 0,C 180,E1 -23994.432,E2 -23994.432} C_VEL
LIN {X 0,Y 159.102,Z 450.556,A -85,B 0,C 180,E1 -23997.989,E2 -23997.989} C_VEL
LIN {X 0,Y 155.62,Z 455.316,A -85,B 0,C 180,E1 -24001.693,E2 -24001.693} C_VEL
LIN {X 0,Y 152.817,Z 458.944,A -85,B 0,C 180,E1 -24005.549,E2 -24005.549} C_VEL
LIN {X 0,Y 151.236,Z 460.903,A -85,B 0,C 180,E1 -24008.344,E2 -24008.344} C_VEL
LIN {X 0,Y 148.987,Z 463.186,A -85,B 0,C 180,E1 -24013.559,E2 -24013.559} C_VEL
LIN {X 0,Y 147.808,Z 463.983,A -85,B 0,C 180,E1 -24019.036,E2 -24019.036} C_VEL
LIN {X 0,Y 147.616,Z 463.751,A -85,B 0,C 180,E1 -24021.788,E2 -24021.788} C_VEL
LIN {X 0,Y 147.626,Z 463.13,A -85,B 0,C 180,E1 -24024.536,E2 -24024.536} C_VEL
LIN {X 0,Y 147.729,Z 462.03,A -85,B 0,C 180,E1 -24027.513,E2 -24027.513} C_VEL
LIN {X 0,Y 147.936,Z 460.735,A -85,B 0,C 180,E1 -24030,E2 -24030} C_VEL
LIN {X 0,Y 148.705,Z 457.817,A -85,B 0,C 180,E1 -24034.065,E2 -24034.065} C_VEL
LIN {X 0,Y 149.931,Z 453.877,A -85,B 0,C 180,E1 -24038.084,E2 -24038.084} C_VEL
LIN {X 0,Y 151.743,Z 448.804,A -85,B 0,C 180,E1 -24042.03,E2 -24042.03} C_VEL
LIN {X 0,Y 154.151,Z 442.417,A -85,B 0,C 180,E1 -24045.876,E2 -24045.876} C_VEL
LIN {X 0,Y 157.222,Z 434.453,A -85,B 0,C 180,E1 -24049.588,E2 -24049.588} C_VEL
LIN {X 0,Y 160.168,Z 426.389,A -85,B 0,C 180,E1 -24052.558,E2 -24052.558} C_VEL
LIN {X 0,Y 163.504,Z 416.442,A -85,B 0,C 180,E1 -24055.457,E2 -24055.457} C_VEL
LIN {X 0,Y 166.763,Z 405.269,A -85,B 0,C 180,E1 -24057.959,E2 -24057.959} C_VEL
LIN {X 0,Y 169.457,Z 394.337,A -85,B 0,C 180,E1 -24059.847,E2 -24059.847} C_VEL
LIN {X 0,Y 171.87,Z 382.24,A -85,B 0,C 180,E1 -24061.424,E2 -24061.424} C_VEL
LIN {X 0,Y 173.758,Z 369.5,A -85,B 0,C 180,E1 -24062.589,E2 -24062.589} C_VEL
LIN {X 0,Y 175.02,Z 356.416,A -85,B 0,C 180,E1 -24063.336,E2 -24063.336} C_VEL
LIN {X 0,Y 177.832,Z 309.039,A -85,B 0,C 180,E1 -24065.042,E2 -24065.042} C_VEL
LIN {X 0,Y 174.532,Z 300.483,A -85,B 0,C 180,E1 -24066.355,E2 -24066.355} C_VEL
LIN {X 0,Y 168.817,Z 289.654,A -85,B 0,C 180,E1 -24068.591,E2 -24068.591} C_VEL
LIN {X 0,Y 162.021,Z 278.442,A -85,B 0,C 180,E1 -24071.473,E2 -24071.473} C_VEL
LIN {X 0,Y 156.254,Z 270.099,A -85,B 0,C 180,E1 -24074.169,E2 -24074.169} C_VEL
LIN {X 0,Y 153.926,Z 266.901,A -85,B 0,C 180,E1 -24075.346,E2 -24075.346} C_VEL
LIN {X 0,Y 153.171,Z 265.766,A -85,B 0,C 180,E1 -24075.748,E2 -24075.748} C_VEL
LIN {X 0,Y 151.126,Z 263.603,A -85,B 0,C 180,E1 -24076.808,E2 -24076.808} C_VEL
LIN {X 0,Y 150.213,Z 261.094,A -85,B 0,C 180,E1 -24077.412,E2 -24077.412} C_VEL
LIN {X 0,Y 150.156,Z 260.781,A -85,B 0,C 180,E1 -24077.495,E2 -24077.495} C_VEL
LIN {X 0,Y 150.18,Z 260.777,A -85,B 0,C 180,E1 -24082.707,E2 -24082.707} C_VEL
LIN {X 0,Y 150.215,Z 260.738,A -85,B 0,C 180,E1 -24087.368,E2 -24087.368} C_VEL
LIN {X 0,Y 150.245,Z 260.769,A -85,B 0,C 180,E1 -24092.718,E2 -24092.718} C_VEL
LIN {X 0,Y 150.352,Z 260.717,A -85,B 0,C 180,E1 -24099.207,E2 -24099.207} C_VEL
LIN {X 0,Y 150.363,Z 260.75,A -85,B 0,C 180,E1 -24103.713,E2 -24103.713} C_VEL
LIN {X 0,Y 150.61,Z 260.672,A -85,B 0,C 180,E1 -24109.242,E2 -24109.242} C_VEL
LIN {X 0,Y 150.684,Z 260.689,A -85,B 0,C 180,E1 -24111.956,E2 -24111.956} C_VEL
LIN {X 0,Y 151.217,Z 260.645,A -85,B 0,C 180,E1 -24120,E2 -24120} C_VEL
LIN {X 0,Y 150.756,Z 260.704,A -85,B 0,C 180,E1 -24128.039,E2 -24128.039} C_VEL
LIN {X 0,Y 150.612,Z 260.702,A -85,B 0,C 180,E1 -24131.502,E2 -24131.502} C_VEL
LIN {X 0,Y 150.331,Z 260.753,A -85,B 0,C 180,E1 -24136.29,E2 -24136.29} C_VEL
LIN {X 0,Y 150.339,Z 260.752,A -85,B 0,C 180,E1 -24140.78,E2 -24140.78} C_VEL
LIN {X 0,Y 150.238,Z 260.77,A -85,B 0,C 180,E1 -24147.277,E2 -24147.277} C_VEL
LIN {X 0,Y 150.208,Z 260.775,A -85,B 0,C 180,E1 -24152.628,E2 -24152.628} C_VEL
LIN {X 0,Y 150.218,Z 260.768,A -85,B 0,C 180,E1 -24156.204,E2 -24156.204} C_VEL
LIN {X 0,Y 151.197,Z 263.616,A -85,B 0,C 180,E1 -24156.872,E2 -24156.872} C_VEL
LIN {X 0,Y 153.21,Z 265.774,A -85,B 0,C 180,E1 -24157.916,E2 -24157.916} C_VEL
LIN {X 0,Y 154.26,Z 267.378,A -85,B 0,C 180,E1 -24158.475,E2 -24158.475} C_VEL
LIN {X 0,Y 156.54,Z 270.385,A -85,B 0,C 180,E1 -24159.61,E2 -24159.61} C_VEL
LIN {X 0,Y 160.1,Z 275.797,A -85,B 0,C 180,E1 -24161.32,E2 -24161.32} C_VEL
LIN {X 0,Y 166.4,Z 287.468,A -85,B 0,C 180,E1 -24164.176,E2 -24164.176} C_VEL
LIN {X 0,Y 171.91,Z 299.832,A -85,B 0,C 180,E1 -24166.525,E2 -24166.525} C_VEL
LIN {X 0,Y 176.332,Z 311.807,A -85,B 0,C 180,E1 -24168.358,E2 -24168.358} C_VEL
LIN {X 0,Y 177.118,Z 322.186,A -85,B 0,C 180,E1 -24169.087,E2 -24169.087} C_VEL
LIN {X 0,Y 174.378,Z 368.17,A -85,B 0,C 180,E1 -24170.797,E2 -24170.797} C_VEL
LIN {X 0,Y 172.824,Z 381.133,A -85,B 0,C 180,E1 -24171.655,E2 -24171.655} C_VEL
LIN {X 0,Y 170.55,Z 394.024,A -85,B 0,C 180,E1 -24172.939,E2 -24172.939} C_VEL
LIN {X 0,Y 167.92,Z 405.32,A -85,B 0,C 180,E1 -24174.499,E2 -24174.499} C_VEL
LIN {X 0,Y 164.673,Z 417.006,A -85,B 0,C 180,E1 -24176.668,E2 -24176.668} C_VEL
LIN {X 0,Y 161.294,Z 427.51,A -85,B 0,C 180,E1 -24179.204,E2 -24179.204} C_VEL
LIN {X 0,Y 158.046,Z 436.965,A -85,B 0,C 180,E1 -24182.166,E2 -24182.166} C_VEL
LIN {X 0,Y 155.414,Z 444.738,A -85,B 0,C 180,E1 -24185.279,E2 -24185.279} C_VEL
LIN {X 0,Y 152.568,Z 452.303,A -85,B 0,C 180,E1 -24189.084,E2 -24189.084} C_VEL
LIN {X 0,Y 150.794,Z 456.997,A -85,B 0,C 180,E1 -24192.024,E2 -24192.024} C_VEL
LIN {X 0,Y 149.21,Z 459.704,A -85,B 0,C 180,E1 -24193.94,E2 -24193.94} C_VEL
LIN {X 0,Y 145.205,Z 463.487,A -85,B 0,C 180,E1 -24197.154,E2 -24197.154} C_VEL
LIN {X 0,Y 142.167,Z 466.012,A -85,B 0,C 180,E1 -24199.921,E2 -24199.921} C_VEL
LIN {X 0,Y 140.829,Z 467.647,A -85,B 0,C 180,E1 -24202.17,E2 -24202.17} C_VEL
LIN {X 0,Y 140.678,Z 468.096,A -85,B 0,C 180,E1 -24202.947,E2 -24202.947} C_VEL
LIN {X 0,Y 140.547,Z 470.263,A -85,B 0,C 180,E1 -24207.134,E2 -24207.134} C_VEL
LIN {X 0,Y 140.569,Z 471.385,A -85,B 0,C 180,E1 -24210.644,E2 -24210.644} C_VEL
LIN {X 0,Y 140.617,Z 471.878,A -85,B 0,C 180,E1 -24215.737,E2 -24215.737} C_VEL
LIN {X 0,Y 141.441,Z 470.932,A -85,B 0,C 180,E1 -24221.464,E2 -24221.464} C_VEL
LIN {X 0,Y 142.304,Z 469.885,A -85,B 0,C 180,E1 -24224.296,E2 -24224.296} C_VEL
LIN {X 0,Y 143.443,Z 468.416,A -85,B 0,C 180,E1 -24227.096,E2 -24227.096} C_VEL
LIN {X 0,Y 145.895,Z 465.42,A -85,B 0,C 180,E1 -24231.179,E2 -24231.179} C_VEL
LIN {X 0,Y 149.029,Z 461.389,A -85,B 0,C 180,E1 -24235.114,E2 -24235.114} C_VEL
LIN {X 0,Y 153.206,Z 455.734,A -85,B 0,C 180,E1 -24239.156,E2 -24239.156} C_VEL
LIN {X 0,Y 157.935,Z 448.5,A -85,B 0,C 180,E1 -24243.033,E2 -24243.033} C_VEL
LIN {X 0,Y 163.079,Z 440.191,A -85,B 0,C 180,E1 -24246.339,E2 -24246.339} C_VEL
LIN {X 0,Y 167.809,Z 431.655,A -85,B 0,C 180,E1 -24248.919,E2 -24248.919} C_VEL
LIN {X 0,Y 172.84,Z 421.14,A -85,B 0,C 180,E1 -24251.358,E2 -24251.358} C_VEL
LIN {X 0,Y 177.176,Z 410.729,A -85,B 0,C 180,E1 -24253.177,E2 -24253.177} C_VEL
LIN {X 0,Y 181.09,Z 399.29,A -85,B 0,C 180,E1 -24254.702,E2 -24254.702} C_VEL
LIN {X 0,Y 184.463,Z 386.179,A -85,B 0,C 180,E1 -24255.983,E2 -24255.983} C_VEL
LIN {X 0,Y 187.016,Z 372.757,A -85,B 0,C 180,E1 -24256.843,E2 -24256.843} C_VEL
LIN {X 0,Y 188.438,Z 359.899,A -85,B 0,C 180,E1 -24257.339,E2 -24257.339} C_VEL
LIN {X 0,Y 190.123,Z 334.75,A -85,B 0,C 180,E1 -24258.191,E2 -24258.191} C_VEL
LIN {X 0,Y 186.09,Z 324.273,A -85,B 0,C 180,E1 -24260.392,E2 -24260.392} C_VEL
LIN {X 0,Y 181.379,Z 313.973,A -85,B 0,C 180,E1 -24263.121,E2 -24263.121} C_VEL
LIN {X 0,Y 176.262,Z 304.007,A -85,B 0,C 180,E1 -24266.413,E2 -24266.413} C_VEL
LIN {X 0,Y 172.874,Z 298.217,A -85,B 0,C 180,E1 -24268.83,E2 -24268.83} C_VEL
LIN {X 0,Y 170.089,Z 293.582,A -85,B 0,C 180,E1 -24271.039,E2 -24271.039} C_VEL
LIN {X 0,Y 167.325,Z 289.588,A -85,B 0,C 180,E1 -24273.439,E2 -24273.439} C_VEL
LIN {X 0,Y 164.621,Z 286.267,A -85,B 0,C 180,E1 -24276.052,E2 -24276.052} C_VEL
LIN {X 0,Y 163.715,Z 284.806,A -85,B 0,C 180,E1 -24277.064,E2 -24277.064} C_VEL
LIN {X 0,Y 161.108,Z 282.189,A -85,B 0,C 180,E1 -24280.134,E2 -24280.134} C_VEL
LIN {X 0,Y 159.855,Z 279.637,A -85,B 0,C 180,E1 -24282.076,E2 -24282.076} C_VEL
LIN {X 0,Y 157.104,Z 277.591,A -85,B 0,C 180,E1 -24286.87,E2 -24286.87} C_VEL
LIN {X 0,Y 155.919,Z 274.855,A -85,B 0,C 180,E1 -24290.603,E2 -24290.603} C_VEL
LIN {X 0,Y 155.69,Z 273.86,A -85,B 0,C 180,E1 -24291.827,E2 -24291.827} C_VEL
LIN {X 0,Y 155.416,Z 273.691,A -85,B 0,C 180,E1 -24301.296,E2 -24301.296} C_VEL
LIN {X 0,Y 155.749,Z 274.047,A -85,B 0,C 180,E1 -24302.91,E2 -24302.91} C_VEL
LIN {X 0,Y 156.801,Z 276.788,A -85,B 0,C 180,E1 -24306.717,E2 -24306.717} C_VEL
LIN {X 0,Y 159.662,Z 279.475,A -85,B 0,C 180,E1 -24312.063,E2 -24312.063} C_VEL
LIN {X 0,Y 160.109,Z 280.113,A -85,B 0,C 180,E1 -24312.759,E2 -24312.759} C_VEL
LIN {X 0,Y 162.235,Z 283.449,A -85,B 0,C 180,E1 -24315.709,E2 -24315.709} C_VEL
LIN {X 0,Y 164.117,Z 285.253,A -85,B 0,C 180,E1 -24317.794,E2 -24317.794} C_VEL
LIN {X 0,Y 166.539,Z 288.758,A -85,B 0,C 180,E1 -24320.28,E2 -24320.28} C_VEL
LIN {X 0,Y 167.931,Z 290.302,A -85,B 0,C 180,E1 -24321.524,E2 -24321.524} C_VEL
LIN {X 0,Y 171.592,Z 295.373,A -85,B 0,C 180,E1 -24324.546,E2 -24324.546} C_VEL
LIN {X 0,Y 175.09,Z 300.504,A -85,B 0,C 180,E1 -24327.087,E2 -24327.087} C_VEL
LIN {X 0,Y 179.097,Z 306.478,A -85,B 0,C 180,E1 -24329.675,E2 -24329.675} C_VEL
LIN {X 0,Y 184.7,Z 315.909,A -85,B 0,C 180,E1 -24332.917,E2 -24332.917} C_VEL
LIN {X 0,Y 187.655,Z 321.638,A -85,B 0,C 180,E1 -24334.5,E2 -24334.5} C_VEL
LIN {X 0,Y 190.624,Z 328.602,A -85,B 0,C 180,E1 -24336.06,E2 -24336.06} C_VEL
LIN {X 0,Y 188.085,Z 361.435,A -85,B 0,C 180,E1 -24337.152,E2 -24337.152} C_VEL
LIN {X 0,Y 186.06,Z 374.979,A -85,B 0,C 180,E1 -24337.954,E2 -24337.954} C_VEL
LIN {X 0,Y 183.261,Z 387.475,A -85,B 0,C 180,E1 -24339.051,E2 -24339.051} C_VEL
LIN {X 0,Y 179.958,Z 398.603,A -85,B 0,C 180,E1 -24340.399,E2 -24340.399} C_VEL
LIN {X 0,Y 175.608,Z 410.178,A -85,B 0,C 180,E1 -24342.236,E2 -24342.236} C_VEL
LIN {X 0,Y 170.891,Z 420.896,A -85,B 0,C 180,E1 -24344.518,E2 -24344.518} C_VEL
LIN {X 0,Y 166.759,Z 429.07,A -85,B 0,C 180,E1 -24346.776,E2 -24346.776} C_VEL
LIN {X 0,Y 162.144,Z 436.863,A -85,B 0,C 180,E1 -24349.446,E2 -24349.446} C_VEL
LIN {X 0,Y 157.303,Z 444.461,A -85,B 0,C 180,E1 -24352.904,E2 -24352.904} C_VEL
LIN {X 0,Y 153.024,Z 450.548,A -85,B 0,C 180,E1 -24356.555,E2 -24356.555} C_VEL
LIN {X 0,Y 149.319,Z 455.352,A -85,B 0,C 180,E1 -24360.383,E2 -24360.383} C_VEL
LIN {X 0,Y 146.292,Z 459.021,A -85,B 0,C 180,E1 -24364.382,E2 -24364.382} C_VEL
LIN {X 0,Y 144.358,Z 461.22,A -85,B 0,C 180,E1 -24367.671,E2 -24367.671} C_VEL
LIN {X 0,Y 142.12,Z 463.339,A -85,B 0,C 180,E1 -24372.74,E2 -24372.74} C_VEL
LIN {X 0,Y 140.763,Z 464.178,A -85,B 0,C 180,E1 -24378.48,E2 -24378.48} C_VEL
LIN {X 0,Y 140.527,Z 463.977,A -85,B 0,C 180,E1 -24381.371,E2 -24381.371} C_VEL
LIN {X 0,Y 140.527,Z 463.373,A -85,B 0,C 180,E1 -24384.259,E2 -24384.259} C_VEL
LIN {X 0,Y 140.661,Z 462.106,A -85,B 0,C 180,E1 -24387.843,E2 -24387.843} C_VEL
LIN {X 0,Y 141.309,Z 459.195,A -85,B 0,C 180,E1 -24392.851,E2 -24392.851} C_VEL
LIN {X 0,Y 142.419,Z 455.651,A -85,B 0,C 180,E1 -24397.086,E2 -24397.086} C_VEL
LIN {X 0,Y 144.136,Z 451.008,A -85,B 0,C 180,E1 -24401.247,E2 -24401.247} C_VEL
LIN {X 0,Y 146.922,Z 444.018,A -85,B 0,C 180,E1 -24405.965,E2 -24405.965} C_VEL
LIN {X 0,Y 149.972,Z 436.452,A -85,B 0,C 180,E1 -24409.862,E2 -24409.862} C_VEL
LIN {X 0,Y 153.3,Z 427.952,A -85,B 0,C 180,E1 -24413.238,E2 -24413.238} C_VEL
LIN {X 0,Y 156.781,Z 418.184,A -85,B 0,C 180,E1 -24416.274,E2 -24416.274} C_VEL
LIN {X 0,Y 160.169,Z 407.478,A -85,B 0,C 180,E1 -24418.859,E2 -24418.859} C_VEL
LIN {X 0,Y 162.981,Z 397.072,A -85,B 0,C 180,E1 -24420.802,E2 -24420.802} C_VEL
LIN {X 0,Y 165.721,Z 384.564,A -85,B 0,C 180,E1 -24422.552,E2 -24422.552} C_VEL
LIN {X 0,Y 167.802,Z 371.772,A -85,B 0,C 180,E1 -24423.837,E2 -24423.837} C_VEL
LIN {X 0,Y 169.211,Z 358.739,A -85,B 0,C 180,E1 -24424.675,E2 -24424.675} C_VEL
LIN {X 0,Y 172.105,Z 310.618,A -85,B 0,C 180,E1 -24426.487,E2 -24426.487} C_VEL
LIN {X 0,Y 169.626,Z 304.221,A -85,B 0,C 180,E1 -24427.541,E2 -24427.541} C_VEL
LIN {X 0,Y 164.444,Z 294.185,A -85,B 0,C 180,E1 -24429.71,E2 -24429.71} C_VEL
LIN {X 0,Y 158.119,Z 283.532,A -85,B 0,C 180,E1 -24432.569,E2 -24432.569} C_VEL
LIN {X 0,Y 152.455,Z 275.295,A -85,B 0,C 180,E1 -24435.388,E2 -24435.388} C_VEL
LIN {X 0,Y 149.592,Z 271.315,A -85,B 0,C 180,E1 -24436.945,E2 -24436.945} C_VEL
LIN {X 0,Y 147.275,Z 268.239,A -85,B 0,C 180,E1 -24438.278,E2 -24438.278} C_VEL
LIN {X 0,Y 146.687,Z 266.978,A -85,B 0,C 180,E1 -24438.667,E2 -24438.667} C_VEL
LIN {X 0,Y 144.296,Z 264.867,A -85,B 0,C 180,E1 -24440.07,E2 -24440.07} C_VEL
LIN {X 0,Y 143.179,Z 262.312,A -85,B 0,C 180,E1 -24440.889,E2 -24440.889} C_VEL
LIN {X 0,Y 143.07,Z 261.657,A -85,B 0,C 180,E1 -24441.069,E2 -24441.069} C_VEL
LIN {X 0,Y 143.182,Z 261.613,A -85,B 0,C 180,E1 -24447.321,E2 -24447.321} C_VEL
LIN {X 0,Y 143.191,Z 261.647,A -85,B 0,C 180,E1 -24452.062,E2 -24452.062} C_VEL
LIN {X 0,Y 143.278,Z 261.593,A -85,B 0,C 180,E1 -24458.745,E2 -24458.745} C_VEL
LIN {X 0,Y 143.303,Z 261.631,A -85,B 0,C 180,E1 -24462.887,E2 -24462.887} C_VEL
LIN {X 0,Y 143.536,Z 261.551,A -85,B 0,C 180,E1 -24468.705,E2 -24468.705} C_VEL
LIN {X 0,Y 143.61,Z 261.561,A -85,B 0,C 180,E1 -24471.557,E2 -24471.557} C_VEL
LIN {X 0,Y 144.175,Z 261.522,A -85,B 0,C 180,E1 -24480,E2 -24480} C_VEL
LIN {X 0,Y 143.674,Z 261.583,A -85,B 0,C 180,E1 -24488.438,E2 -24488.438} C_VEL
LIN {X 0,Y 143.548,Z 261.582,A -85,B 0,C 180,E1 -24491.712,E2 -24491.712} C_VEL
LIN {X 0,Y 143.269,Z 261.625,A -85,B 0,C 180,E1 -24497.117,E2 -24497.117} C_VEL
LIN {X 0,Y 143.267,Z 261.637,A -85,B 0,C 180,E1 -24501.244,E2 -24501.244} C_VEL
LIN {X 0,Y 143.183,Z 261.65,A -85,B 0,C 180,E1 -24507.931,E2 -24507.931} C_VEL
LIN {X 0,Y 143.16,Z 261.653,A -85,B 0,C 180,E1 -24512.684,E2 -24512.684} C_VEL
LIN {X 0,Y 143.979,Z 264.214,A -85,B 0,C 180,E1 -24513.352,E2 -24513.352} C_VEL
LIN {X 0,Y 145.868,Z 266.401,A -85,B 0,C 180,E1 -24514.52,E2 -24514.52} C_VEL
LIN {X 0,Y 146.922,Z 267.321,A -85,B 0,C 180,E1 -24515.123,E2 -24515.123} C_VEL
LIN {X 0,Y 148.879,Z 270.532,A -85,B 0,C 180,E1 -24516.311,E2 -24516.311} C_VEL
LIN {X 0,Y 150.595,Z 272.557,A -85,B 0,C 180,E1 -24517.248,E2 -24517.248} C_VEL
LIN {X 0,Y 154.277,Z 277.909,A -85,B 0,C 180,E1 -24519.203,E2 -24519.203} C_VEL
LIN {X 0,Y 156.435,Z 281.295,A -85,B 0,C 180,E1 -24520.29,E2 -24520.29} C_VEL
LIN {X 0,Y 162.01,Z 291.851,A -85,B 0,C 180,E1 -24522.985,E2 -24522.985} C_VEL
LIN {X 0,Y 167.102,Z 303.666,A -85,B 0,C 180,E1 -24525.32,E2 -24525.32} C_VEL
LIN {X 0,Y 171.016,Z 314.652,A -85,B 0,C 180,E1 -24527.07,E2 -24527.07} C_VEL
LIN {X 0,Y 171.508,Z 323.351,A -85,B 0,C 180,E1 -24527.671,E2 -24527.671} C_VEL
LIN {X 0,Y 168.663,Z 368.574,A -85,B 0,C 180,E1 -24529.4,E2 -24529.4} C_VEL
LIN {X 0,Y 167.105,Z 380.977,A -85,B 0,C 180,E1 -24530.244,E2 -24530.244} C_VEL
LIN {X 0,Y 164.911,Z 392.946,A -85,B 0,C 180,E1 -24531.445,E2 -24531.445} C_VEL
LIN {X 0,Y 162.185,Z 404.485,A -85,B 0,C 180,E1 -24533.041,E2 -24533.041} C_VEL
LIN {X 0,Y 158.782,Z 416.308,A -85,B 0,C 180,E1 -24535.259,E2 -24535.259} C_VEL
LIN {X 0,Y 155.223,Z 426.898,A -85,B 0,C 180,E1 -24537.859,E2 -24537.859} C_VEL
LIN {X 0,Y 151.743,Z 436.44,A -85,B 0,C 180,E1 -24540.902,E2 -24540.902} C_VEL
LIN {X 0,Y 148.797,Z 444.615,A -85,B 0,C 180,E1 -24544.287,E2 -24544.287} C_VEL
LIN {X 0,Y 145.89,Z 451.887,A -85,B 0,C 180,E1 -24548.078,E2 -24548.078} C_VEL
LIN {X 0,Y 143.134,Z 458.925,A -85,B 0,C 180,E1 -24552.866,E2 -24552.866} C_VEL
LIN {X 0,Y 141.698,Z 463.588,A -85,B 0,C 180,E1 -24557.103,E2 -24557.103} C_VEL
LIN {X 0,Y 140.851,Z 467.127,A -85,B 0,C 180,E1 -24561.391,E2 -24561.391} C_VEL
LIN {X 0,Y 140.678,Z 468.096,A -85,B 0,C 180,E1 -24562.947,E2 -24562.947} C_VEL
LIN {X 0,Y 140.255,Z 469.031,A -85,B 0,C 180,E1 -24564.502,E2 -24564.502} C_VEL
LIN {X 0,Y 138.793,Z 470.117,A -85,B 0,C 180,E1 -24566.821,E2 -24566.821} C_VEL
LIN {X 0,Y 134.456,Z 471.476,A -85,B 0,C 180,E1 -24572.39,E2 -24572.39} C_VEL
LIN {X 0,Y 133.541,Z 471.664,A -85,B 0,C 180,E1 -24574.93,E2 -24574.93} C_VEL
LIN {X 0,Y 133.522,Z 471.676,A -85,B 0,C 180,E1 -24575.789,E2 -24575.789} C_VEL
LIN {X 0,Y 133.84,Z 471.421,A -85,B 0,C 180,E1 -24579.064,E2 -24579.064} C_VEL
LIN {X 0,Y 135.409,Z 469.742,A -85,B 0,C 180,E1 -24585.041,E2 -24585.041} C_VEL
LIN {X 0,Y 136.638,Z 468.304,A -85,B 0,C 180,E1 -24587.976,E2 -24587.976} C_VEL
LIN {X 0,Y 139.277,Z 465.336,A -85,B 0,C 180,E1 -24592.238,E2 -24592.238} C_VEL
LIN {X 0,Y 142.621,Z 461.339,A -85,B 0,C 180,E1 -24596.327,E2 -24596.327} C_VEL
LIN {X 0,Y 147.346,Z 455.213,A -85,B 0,C 180,E1 -24600.846,E2 -24600.846} C_VEL
LIN {X 0,Y 152.012,Z 448.546,A -85,B 0,C 180,E1 -24604.497,E2 -24604.497} C_VEL
LIN {X 0,Y 157.413,Z 440.29,A -85,B 0,C 180,E1 -24607.872,E2 -24607.872} C_VEL
LIN {X 0,Y 162.351,Z 431.835,A -85,B 0,C 180,E1 -24610.491,E2 -24610.491} C_VEL
LIN {X 0,Y 167.595,Z 421.404,A -85,B 0,C 180,E1 -24612.956,E2 -24612.956} C_VEL
LIN {X 0,Y 172.087,Z 411.092,A -85,B 0,C 180,E1 -24614.788,E2 -24614.788} C_VEL
LIN {X 0,Y 176.14,Z 399.801,A -85,B 0,C 180,E1 -24616.319,E2 -24616.319} C_VEL
LIN {X 0,Y 179.346,Z 388.29,A -85,B 0,C 180,E1 -24617.494,E2 -24617.494} C_VEL
LIN {X 0,Y 182.111,Z 374.758,A -85,B 0,C 180,E1 -24618.429,E2 -24618.429} C_VEL
LIN {X 0,Y 183.79,Z 361.828,A -85,B 0,C 180,E1 -24618.969,E2 -24618.969} C_VEL
LIN {X 0,Y 185.529,Z 337.08,A -85,B 0,C 180,E1 -24619.818,E2 -24619.818} C_VEL
LIN {X 0,Y 181.762,Z 327.211,A -85,B 0,C 180,E1 -24622.046,E2 -24622.046} C_VEL
LIN {X 0,Y 177.357,Z 317.353,A -85,B 0,C 180,E1 -24624.829,E2 -24624.829} C_VEL
LIN {X 0,Y 172.73,Z 308.31,A -85,B 0,C 180,E1 -24628.066,E2 -24628.066} C_VEL
LIN {X 0,Y 169.561,Z 302.61,A -85,B 0,C 180,E1 -24630.557,E2 -24630.557} C_VEL
LIN {X 0,Y 167.336,Z 298.851,A -85,B 0,C 180,E1 -24632.484,E2 -24632.484} C_VEL
LIN {X 0,Y 165.438,Z 296.031,A -85,B 0,C 180,E1 -24634.25,E2 -24634.25} C_VEL
LIN {X 0,Y 162.745,Z 292.523,A -85,B 0,C 180,E1 -24637.024,E2 -24637.024} C_VEL
LIN {X 0,Y 161.896,Z 291.321,A -85,B 0,C 180,E1 -24638.012,E2 -24638.012} C_VEL
LIN {X 0,Y 159.546,Z 288.647,A -85,B 0,C 180,E1 -24641.005,E2 -24641.005} C_VEL
LIN {X 0,Y 158.384,Z 286.449,A -85,B 0,C 180,E1 -24642.904,E2 -24642.904} C_VEL
LIN {X 0,Y 155.739,Z 284.094,A -85,B 0,C 180,E1 -24648.045,E2 -24648.045} C_VEL
LIN {X 0,Y 154.74,Z 280.865,A -85,B 0,C 180,E1 -24652.169,E2 -24652.169} C_VEL
LIN {X 0,Y 154.725,Z 280.779,A -85,B 0,C 180,E1 -24662.15,E2 -24662.15} C_VEL
LIN {X 0,Y 155.77,Z 283.756,A -85,B 0,C 180,E1 -24666.355,E2 -24666.355} C_VEL
LIN {X 0,Y 158.674,Z 286.741,A -85,B 0,C 180,E1 -24671.976,E2 -24671.976} C_VEL
LIN {X 0,Y 160.72,Z 290.119,A -85,B 0,C 180,E1 -24675.008,E2 -24675.008} C_VEL
LIN {X 0,Y 162.439,Z 291.839,A -85,B 0,C 180,E1 -24677.021,E2 -24677.021} C_VEL
LIN {X 0,Y 164.87,Z 295.403,A -85,B 0,C 180,E1 -24679.638,E2 -24679.638} C_VEL
LIN {X 0,Y 166.248,Z 297.169,A -85,B 0,C 180,E1 -24680.943,E2 -24680.943} C_VEL
LIN {X 0,Y 169.325,Z 301.508,A -85,B 0,C 180,E1 -24683.608,E2 -24683.608} C_VEL
LIN {X 0,Y 172.452,Z 306.224,A -85,B 0,C 180,E1 -24686.02,E2 -24686.02} C_VEL
LIN {X 0,Y 176.639,Z 312.84,A -85,B 0,C 180,E1 -24688.891,E2 -24688.891} C_VEL
LIN {X 0,Y 181.456,Z 321.197,A -85,B 0,C 180,E1 -24691.836,E2 -24691.836} C_VEL
LIN {X 0,Y 184.184,Z 326.723,A -85,B 0,C 180,E1 -24693.398,E2 -24693.398} C_VEL
LIN {X 0,Y 186.04,Z 331.22,A -85,B 0,C 180,E1 -24694.448,E2 -24694.448} C_VEL
LIN {X 0,Y 183.531,Z 362.07,A -85,B 0,C 180,E1 -24695.489,E2 -24695.489} C_VEL
LIN {X 0,Y 181.443,Z 375.341,A -85,B 0,C 180,E1 -24696.279,E2 -24696.279} C_VEL
LIN {X 0,Y 178.55,Z 387.785,A -85,B 0,C 180,E1 -24697.381,E2 -24697.381} C_VEL
LIN {X 0,Y 174.846,Z 399.685,A -85,B 0,C 180,E1 -24698.85,E2 -24698.85} C_VEL
LIN {X 0,Y 170.318,Z 411.095,A -85,B 0,C 180,E1 -24700.692,E2 -24700.692} C_VEL
LIN {X 0,Y 165.519,Z 421.456,A -85,B 0,C 180,E1 -24702.955,E2 -24702.955} C_VEL
LIN {X 0,Y 160.604,Z 430.549,A -85,B 0,C 180,E1 -24705.56,E2 -24705.56} C_VEL
LIN {X 0,Y 154.953,Z 439.48,A -85,B 0,C 180,E1 -24708.878,E2 -24708.878} C_VEL
LIN {X 0,Y 150.043,Z 446.635,A -85,B 0,C 180,E1 -24712.488,E2 -24712.488} C_VEL
LIN {X 0,Y 145.688,Z 452.309,A -85,B 0,C 180,E1 -24716.306,E2 -24716.306} C_VEL
LIN {X 0,Y 141.924,Z 456.759,A -85,B 0,C 180,E1 -24720.317,E2 -24720.317} C_VEL
LIN {X 0,Y 139.828,Z 459.1,A -85,B 0,C 180,E1 -24723.105,E2 -24723.105} C_VEL
LIN {X 0,Y 137.53,Z 461.52,A -85,B 0,C 180,E1 -24726.902,E2 -24726.902} C_VEL
LIN {X 0,Y 135.291,Z 463.492,A -85,B 0,C 180,E1 -24731.839,E2 -24731.839} C_VEL
LIN {X 0,Y 133.745,Z 464.367,A -85,B 0,C 180,E1 -24737.866,E2 -24737.866} C_VEL
LIN {X 0,Y 133.461,Z 464.202,A -85,B 0,C 180,E1 -24740.91,E2 -24740.91} C_VEL
LIN {X 0,Y 133.424,Z 463.616,A -85,B 0,C 180,E1 -24743.953,E2 -24743.953} C_VEL
LIN {X 0,Y 133.598,Z 462.157,A -85,B 0,C 180,E1 -24748.219,E2 -24748.219} C_VEL
LIN {X 0,Y 134.582,Z 458.449,A -85,B 0,C 180,E1 -24754.493,E2 -24754.493} C_VEL
LIN {X 0,Y 135.92,Z 454.59,A -85,B 0,C 180,E1 -24758.924,E2 -24758.924} C_VEL
LIN {X 0,Y 137.961,Z 449.606,A -85,B 0,C 180,E1 -24763.252,E2 -24763.252} C_VEL
LIN {X 0,Y 140.59,Z 443.352,A -85,B 0,C 180,E1 -24767.454,E2 -24767.454} C_VEL
LIN {X 0,Y 143.976,Z 435.512,A -85,B 0,C 180,E1 -24771.475,E2 -24771.475} C_VEL
LIN {X 0,Y 147.874,Z 425.76,A -85,B 0,C 180,E1 -24775.324,E2 -24775.324} C_VEL
LIN {X 0,Y 151.642,Z 415.588,A -85,B 0,C 180,E1 -24778.362,E2 -24778.362} C_VEL
LIN {X 0,Y 155.251,Z 404.103,A -85,B 0,C 180,E1 -24780.993,E2 -24780.993} C_VEL
LIN {X 0,Y 158.272,Z 392.792,A -85,B 0,C 180,E1 -24782.953,E2 -24782.953} C_VEL
LIN {X 0,Y 160.693,Z 381.187,A -85,B 0,C 180,E1 -24784.46,E2 -24784.46} C_VEL
LIN {X 0,Y 162.707,Z 368.066,A -85,B 0,C 180,E1 -24785.645,E2 -24785.645} C_VEL
LIN {X 0,Y 163.937,Z 355.793,A -85,B 0,C 180,E1 -24786.33,E2 -24786.33} C_VEL
LIN {X 0,Y 166.616,Z 312.537,A -85,B 0,C 180,E1 -24787.974,E2 -24787.974} C_VEL
LIN {X 0,Y 164.334,Z 306.972,A -85,B 0,C 180,E1 -24788.999,E2 -24788.999} C_VEL
LIN {X 0,Y 159.027,Z 296.714,A -85,B 0,C 180,E1 -24791.404,E2 -24791.404} C_VEL
LIN {X 0,Y 153.665,Z 287.757,A -85,B 0,C 180,E1 -24794.026,E2 -24794.026} C_VEL
LIN {X 0,Y 148.803,Z 280.473,A -85,B 0,C 180,E1 -24796.633,E2 -24796.633} C_VEL
LIN {X 0,Y 146.245,Z 276.893,A -85,B 0,C 180,E1 -24798.117,E2 -24798.117} C_VEL
LIN {X 0,Y 143.7,Z 273.183,A -85,B 0,C 180,E1 -24799.707,E2 -24799.707} C_VEL
LIN {X 0,Y 140.834,Z 269.867,A -85,B 0,C 180,E1 -24801.571,E2 -24801.571} C_VEL
LIN {X 0,Y 139.87,Z 267.988,A -85,B 0,C 180,E1 -24802.304,E2 -24802.304} C_VEL
LIN {X 0,Y 137.462,Z 265.992,A -85,B 0,C 180,E1 -24803.987,E2 -24803.987} C_VEL
LIN {X 0,Y 136.285,Z 263.699,A -85,B 0,C 180,E1 -24804.991,E2 -24804.991} C_VEL
LIN {X 0,Y 136.044,Z 262.516,A -85,B 0,C 180,E1 -24805.371,E2 -24805.371} C_VEL
LIN {X 0,Y 136.117,Z 262.523,A -85,B 0,C 180,E1 -24811.372,E2 -24811.372} C_VEL
LIN {X 0,Y 136.245,Z 262.468,A -85,B 0,C 180,E1 -24818.833,E2 -24818.833} C_VEL
LIN {X 0,Y 136.269,Z 262.49,A -85,B 0,C 180,E1 -24825.056,E2 -24825.056} C_VEL
LIN {X 0,Y 136.431,Z 262.435,A -85,B 0,C 180,E1 -24828.166,E2 -24828.166} C_VEL
LIN {X 0,Y 136.539,Z 262.434,A -85,B 0,C 180,E1 -24831.117,E2 -24831.117} C_VEL
LIN {X 0,Y 137.132,Z 262.399,A -85,B 0,C 180,E1 -24840,E2 -24840} C_VEL
LIN {X 0,Y 136.599,Z 262.459,A -85,B 0,C 180,E1 -24848.879,E2 -24848.879} C_VEL
LIN {X 0,Y 136.475,Z 262.462,A -85,B 0,C 180,E1 -24851.921,E2 -24851.921} C_VEL
LIN {X 0,Y 136.188,Z 262.501,A -85,B 0,C 180,E1 -24858.037,E2 -24858.037} C_VEL
LIN {X 0,Y 136.189,Z 262.52,A -85,B 0,C 180,E1 -24861.739,E2 -24861.739} C_VEL
LIN {X 0,Y 136.105,Z 262.555,A -85,B 0,C 180,E1 -24868.42,E2 -24868.42} C_VEL
LIN {X 0,Y 136.904,Z 265.089,A -85,B 0,C 180,E1 -24869.207,E2 -24869.207} C_VEL
LIN {X 0,Y 138.8,Z 267.319,A -85,B 0,C 180,E1 -24870.631,E2 -24870.631} C_VEL
LIN {X 0,Y 140.172,Z 268.356,A -85,B 0,C 180,E1 -24871.555,E2 -24871.555} C_VEL
LIN {X 0,Y 142.013,Z 271.412,A -85,B 0,C 180,E1 -24872.876,E2 -24872.876} C_VEL
LIN {X 0,Y 143.949,Z 273.518,A -85,B 0,C 180,E1 -24874.097,E2 -24874.097} C_VEL
LIN {X 0,Y 146.527,Z 277.144,A -85,B 0,C 180,E1 -24875.687,E2 -24875.687} C_VEL
LIN {X 0,Y 150.724,Z 283.276,A -85,B 0,C 180,E1 -24878.074,E2 -24878.074} C_VEL
LIN {X 0,Y 152.589,Z 286.317,A -85,B 0,C 180,E1 -24879.081,E2 -24879.081} C_VEL
LIN {X 0,Y 157.825,Z 296.629,A -85,B 0,C 180,E1 -24881.802,E2 -24881.802} C_VEL
LIN {X 0,Y 162.442,Z 307.668,A -85,B 0,C 180,E1 -24884.076,E2 -24884.076} C_VEL
LIN {X 0,Y 165.642,Z 316.768,A -85,B 0,C 180,E1 -24885.615,E2 -24885.615} C_VEL
LIN {X 0,Y 166.08,Z 323.1,A -85,B 0,C 180,E1 -24886.105,E2 -24886.105} C_VEL
LIN {X 0,Y 163.158,Z 368.083,A -85,B 0,C 180,E1 -24887.857,E2 -24887.857} C_VEL
LIN {X 0,Y 161.426,Z 381.238,A -85,B 0,C 180,E1 -24888.77,E2 -24888.77} C_VEL
LIN {X 0,Y 159.161,Z 392.998,A -85,B 0,C 180,E1 -24889.982,E2 -24889.982} C_VEL
LIN {X 0,Y 156.092,Z 405.285,A -85,B 0,C 180,E1 -24891.751,E2 -24891.751} C_VEL
LIN {X 0,Y 152.546,Z 416.905,A -85,B 0,C 180,E1 -24894.027,E2 -24894.027} C_VEL
LIN {X 0,Y 148.831,Z 427.359,A -85,B 0,C 180,E1 -24896.705,E2 -24896.705} C_VEL
LIN {X 0,Y 145.521,Z 435.903,A -85,B 0,C 180,E1 -24899.529,E2 -24899.529} C_VEL
LIN {X 0,Y 142.465,Z 443.788,A -85,B 0,C 180,E1 -24902.85,E2 -24902.85} C_VEL
LIN {X 0,Y 139.749,Z 450.323,A -85,B 0,C 180,E1 -24906.277,E2 -24906.277} C_VEL
LIN {X 0,Y 137.105,Z 456.727,A -85,B 0,C 180,E1 -24910.538,E2 -24910.538} C_VEL
LIN {X 0,Y 135.206,Z 461.813,A -85,B 0,C 180,E1 -24914.936,E2 -24914.936} C_VEL
LIN {X 0,Y 134.079,Z 465.753,A -85,B 0,C 180,E1 -24919.429,E2 -24919.429} C_VEL
LIN {X 0,Y 133.539,Z 468.648,A -85,B 0,C 180,E1 -24923.958,E2 -24923.958} C_VEL
LIN {X 0,Y 133.466,Z 470.013,A -85,B 0,C 180,E1 -24926.982,E2 -24926.982} C_VEL
LIN {X 0,Y 133.532,Z 470.976,A -85,B 0,C 180,E1 -24930,E2 -24930} C_VEL
LIN {X 0,Y 133.46,Z 471.538,A -85,B 0,C 180,E1 -24933.019,E2 -24933.019} C_VEL
LIN {X 0,Y 133.522,Z 471.676,A -85,B 0,C 180,E1 -24935.789,E2 -24935.789} C_VEL
LIN {X 0,Y 133.115,Z 471.641,A -85,B 0,C 180,E1 -24938.322,E2 -24938.322} C_VEL
LIN {X 0,Y 131.021,Z 470.904,A -85,B 0,C 180,E1 -24942.524,E2 -24942.524} C_VEL
LIN {X 0,Y 129.535,Z 469.316,A -85,B 0,C 180,E1 -24946.802,E2 -24946.802} C_VEL
LIN {X 0,Y 130.085,Z 467.948,A -85,B 0,C 180,E1 -24949.338,E2 -24949.338} C_VEL
LIN {X 0,Y 133.857,Z 464.023,A -85,B 0,C 180,E1 -24954.837,E2 -24954.837} C_VEL
LIN {X 0,Y 137.688,Z 459.7,A -85,B 0,C 180,E1 -24959.006,E2 -24959.006} C_VEL
LIN {X 0,Y 142.869,Z 453.19,A -85,B 0,C 180,E1 -24963.601,E2 -24963.601} C_VEL
LIN {X 0,Y 148.014,Z 446.06,A -85,B 0,C 180,E1 -24967.258,E2 -24967.258} C_VEL
LIN {X 0,Y 153.902,Z 437.204,A -85,B 0,C 180,E1 -24970.597,E2 -24970.597} C_VEL
LIN {X 0,Y 159.191,Z 428.132,A -85,B 0,C 180,E1 -24973.18,E2 -24973.18} C_VEL
LIN {X 0,Y 163.618,Z 419.327,A -85,B 0,C 180,E1 -24975.132,E2 -24975.132} C_VEL
LIN {X 0,Y 168.31,Z 408.573,A -85,B 0,C 180,E1 -24976.948,E2 -24976.948} C_VEL
LIN {X 0,Y 172.56,Z 396.509,A -85,B 0,C 180,E1 -24978.45,E2 -24978.45} C_VEL
LIN {X 0,Y 175.971,Z 383.601,A -85,B 0,C 180,E1 -24979.639,E2 -24979.639} C_VEL
LIN {X 0,Y 178.347,Z 371.206,A -85,B 0,C 180,E1 -24980.369,E2 -24980.369} C_VEL
LIN {X 0,Y 179.942,Z 355.733,A -85,B 0,C 180,E1 -24980.947,E2 -24980.947} C_VEL
LIN {X 0,Y 181.097,Z 339.511,A -85,B 0,C 180,E1 -24981.519,E2 -24981.519} C_VEL
LIN {X 0,Y 177.8,Z 330.761,A -85,B 0,C 180,E1 -24983.636,E2 -24983.636} C_VEL
LIN {X 0,Y 173.985,Z 321.988,A -85,B 0,C 180,E1 -24986.248,E2 -24986.248} C_VEL
LIN {X 0,Y 170.091,Z 313.995,A -85,B 0,C 180,E1 -24989.189,E2 -24989.189} C_VEL
LIN {X 0,Y 167.465,Z 309.025,A -85,B 0,C 180,E1 -24991.392,E2 -24991.392} C_VEL
LIN {X 0,Y 165.214,Z 304.988,A -85,B 0,C 180,E1 -24993.469,E2 -24993.469} C_VEL
LIN {X 0,Y 163.448,Z 302.335,A -85,B 0,C 180,E1 -24995.214,E2 -24995.214} C_VEL
LIN {X 0,Y 160.873,Z 298.693,A -85,B 0,C 180,E1 -24998.076,E2 -24998.076} C_VEL
LIN {X 0,Y 157.754,Z 294.646,A -85,B 0,C 180,E1 -25002.332,E2 -25002.332} C_VEL
LIN {X 0,Y 157.047,Z 293.279,A -85,B 0,C 180,E1 -25003.591,E2 -25003.591} C_VEL
LIN {X 0,Y 154.603,Z 290.865,A -85,B 0,C 180,E1 -25008.741,E2 -25008.741} C_VEL
LIN {X 0,Y 153.737,Z 287.89,A -85,B 0,C 180,E1 -25012.778,E2 -25012.778} C_VEL
LIN {X 0,Y 153.764,Z 287.816,A -85,B 0,C 180,E1 -25021.737,E2 -25021.737} C_VEL
LIN {X 0,Y 155.052,Z 291.245,A -85,B 0,C 180,E1 -25026.834,E2 -25026.834} C_VEL
LIN {X 0,Y 157.371,Z 293.642,A -85,B 0,C 180,E1 -25031.377,E2 -25031.377} C_VEL
LIN {X 0,Y 159.55,Z 297.135,A -85,B 0,C 180,E1 -25034.713,E2 -25034.713} C_VEL
LIN {X 0,Y 160.825,Z 298.515,A -85,B 0,C 180,E1 -25036.278,E2 -25036.278} C_VEL
LIN {X 0,Y 163.539,Z 302.411,A -85,B 0,C 180,E1 -25039.299,E2 -25039.299} C_VEL
LIN {X 0,Y 167.271,Z 307.908,A -85,B 0,C 180,E1 -25042.789,E2 -25042.789} C_VEL
LIN {X 0,Y 171.591,Z 314.619,A -85,B 0,C 180,E1 -25046.212,E2 -25046.212} C_VEL
LIN {X 0,Y 176.642,Z 323.413,A -85,B 0,C 180,E1 -25049.684,E2 -25049.684} C_VEL
LIN {X 0,Y 180.248,Z 330.575,A -85,B 0,C 180,E1 -25051.926,E2 -25051.926} C_VEL
LIN {X 0,Y 181.563,Z 333.806,A -85,B 0,C 180,E1 -25052.732,E2 -25052.732} C_VEL
LIN {X 0,Y 179.216,Z 362.065,A -85,B 0,C 180,E1 -25053.71,E2 -25053.71} C_VEL
LIN {X 0,Y 177.036,Z 375.406,A -85,B 0,C 180,E1 -25054.491,E2 -25054.491} C_VEL
LIN {X 0,Y 173.979,Z 388.155,A -85,B 0,C 180,E1 -25055.629,E2 -25055.629} C_VEL
LIN {X 0,Y 169.854,Z 400.766,A -85,B 0,C 180,E1 -25057.203,E2 -25057.203} C_VEL
LIN {X 0,Y 165.171,Z 412.012,A -85,B 0,C 180,E1 -25059.056,E2 -25059.056} C_VEL
LIN {X 0,Y 160.312,Z 421.937,A -85,B 0,C 180,E1 -25061.268,E2 -25061.268} C_VEL
LIN {X 0,Y 155.581,Z 430.382,A -85,B 0,C 180,E1 -25063.717,E2 -25063.717} C_VEL
LIN {X 0,Y 150.551,Z 438.012,A -85,B 0,C 180,E1 -25066.484,E2 -25066.484} C_VEL
LIN {X 0,Y 145.217,Z 445.475,A -85,B 0,C 180,E1 -25070.114,E2 -25070.114} C_VEL
LIN {X 0,Y 141.21,Z 450.538,A -85,B 0,C 180,E1 -25073.328,E2 -25073.328} C_VEL
LIN {X 0,Y 136.985,Z 455.428,A -85,B 0,C 180,E1 -25077.405,E2 -25077.405} C_VEL
LIN {X 0,Y 133.426,Z 459.179,A -85,B 0,C 180,E1 -25081.702,E2 -25081.702} C_VEL
LIN {X 0,Y 130.711,Z 461.829,A -85,B 0,C 180,E1 -25086.072,E2 -25086.072} C_VEL
LIN {X 0,Y 128.487,Z 463.645,A -85,B 0,C 180,E1 -25090.841,E2 -25090.841} C_VEL
LIN {X 0,Y 126.753,Z 464.556,A -85,B 0,C 180,E1 -25097.186,E2 -25097.186} C_VEL
LIN {X 0,Y 126.385,Z 464.424,A -85,B 0,C 180,E1 -25100.397,E2 -25100.397} C_VEL
LIN {X 0,Y 126.311,Z 463.859,A -85,B 0,C 180,E1 -25103.611,E2 -25103.611} C_VEL
LIN {X 0,Y 126.536,Z 462.156,A -85,B 0,C 180,E1 -25108.729,E2 -25108.729} C_VEL
LIN {X 0,Y 127.504,Z 458.764,A -85,B 0,C 180,E1 -25114.743,E2 -25114.743} C_VEL
LIN {X 0,Y 128.93,Z 454.944,A -85,B 0,C 180,E1 -25119.412,E2 -25119.412} C_VEL
LIN {X 0,Y 131.078,Z 450.003,A -85,B 0,C 180,E1 -25123.962,E2 -25123.962} C_VEL
LIN {X 0,Y 133.858,Z 443.8,A -85,B 0,C 180,E1 -25128.362,E2 -25128.362} C_VEL
LIN {X 0,Y 137.423,Z 436.037,A -85,B 0,C 180,E1 -25132.554,E2 -25132.554} C_VEL
LIN {X 0,Y 141.042,Z 427.6,A -85,B 0,C 180,E1 -25136.081,E2 -25136.081} C_VEL
LIN {X 0,Y 145.066,Z 417.397,A -85,B 0,C 180,E1 -25139.375,E2 -25139.375} C_VEL
LIN {X 0,Y 148.805,Z 406.349,A -85,B 0,C 180,E1 -25142.095,E2 -25142.095} C_VEL
LIN {X 0,Y 152.406,Z 393.77,A -85,B 0,C 180,E1 -25144.395,E2 -25144.395} C_VEL
LIN {X 0,Y 155.16,Z 381.245,A -85,B 0,C 180,E1 -25146.074,E2 -25146.074} C_VEL
LIN {X 0,Y 157.271,Z 368.069,A -85,B 0,C 180,E1 -25147.278,E2 -25147.278} C_VEL
LIN {X 0,Y 158.571,Z 355.453,A -85,B 0,C 180,E1 -25147.985,E2 -25147.985} C_VEL
LIN {X 0,Y 161.242,Z 314.511,A -85,B 0,C 180,E1 -25149.558,E2 -25149.558} C_VEL
LIN {X 0,Y 156.678,Z 304.768,A -85,B 0,C 180,E1 -25151.747,E2 -25151.747} C_VEL
LIN {X 0,Y 150.687,Z 294.038,A -85,B 0,C 180,E1 -25154.828,E2 -25154.828} C_VEL
LIN {X 0,Y 145.209,Z 285.651,A -85,B 0,C 180,E1 -25157.948,E2 -25157.948} C_VEL
LIN {X 0,Y 142.425,Z 281.745,A -85,B 0,C 180,E1 -25159.685,E2 -25159.685} C_VEL
LIN {X 0,Y 140.008,Z 278.306,A -85,B 0,C 180,E1 -25161.315,E2 -25161.315} C_VEL
LIN {X 0,Y 137.538,Z 274.947,A -85,B 0,C 180,E1 -25163.1,E2 -25163.1} C_VEL
LIN {X 0,Y 136.678,Z 273.877,A -85,B 0,C 180,E1 -25163.748,E2 -25163.748} C_VEL
LIN {X 0,Y 134.206,Z 271.015,A -85,B 0,C 180,E1 -25165.704,E2 -25165.704} C_VEL
LIN {X 0,Y 133.311,Z 269.071,A -85,B 0,C 180,E1 -25166.554,E2 -25166.554} C_VEL
LIN {X 0,Y 130.769,Z 267.247,A -85,B 0,C 180,E1 -25168.738,E2 -25168.738} C_VEL
LIN {X 0,Y 129.376,Z 264.895,A -85,B 0,C 180,E1 -25170.207,E2 -25170.207} C_VEL
LIN {X 0,Y 129.035,Z 263.395,A -85,B 0,C 180,E1 -25170.782,E2 -25170.782} C_VEL
LIN {X 0,Y 129.031,Z 263.393,A -85,B 0,C 180,E1 -25174.167,E2 -25174.167} C_VEL
LIN {X 0,Y 129.108,Z 263.353,A -85,B 0,C 180,E1 -25177.727,E2 -25177.727} C_VEL
LIN {X 0,Y 129.154,Z 263.372,A -85,B 0,C 180,E1 -25180.943,E2 -25180.943} C_VEL
LIN {X 0,Y 129.389,Z 263.312,A -85,B 0,C 180,E1 -25187.877,E2 -25187.877} C_VEL
LIN {X 0,Y 129.465,Z 263.307,A -85,B 0,C 180,E1 -25190.627,E2 -25190.627} C_VEL
LIN {X 0,Y 130.087,Z 263.276,A -85,B 0,C 180,E1 -25200,E2 -25200} C_VEL
LIN {X 0,Y 129.523,Z 263.334,A -85,B 0,C 180,E1 -25209.368,E2 -25209.368} C_VEL
LIN {X 0,Y 129.355,Z 263.352,A -85,B 0,C 180,E1 -25212.552,E2 -25212.552} C_VEL
LIN {X 0,Y 129.113,Z 263.382,A -85,B 0,C 180,E1 -25219.062,E2 -25219.062} C_VEL
LIN {X 0,Y 129.065,Z 263.402,A -85,B 0,C 180,E1 -25222.934,E2 -25222.934} C_VEL
LIN {X 0,Y 129.828,Z 265.88,A -85,B 0,C 180,E1 -25223.954,E2 -25223.954} C_VEL
LIN {X 0,Y 131.643,Z 268.056,A -85,B 0,C 180,E1 -25225.707,E2 -25225.707} C_VEL
LIN {X 0,Y 133.454,Z 269.324,A -85,B 0,C 180,E1 -25227.226,E2 -25227.226} C_VEL
LIN {X 0,Y 135.221,Z 272.439,A -85,B 0,C 180,E1 -25228.793,E2 -25228.793} C_VEL
LIN {X 0,Y 137.537,Z 274.795,A -85,B 0,C 180,E1 -25230.532,E2 -25230.532} C_VEL
LIN {X 0,Y 140.022,Z 278.252,A -85,B 0,C 180,E1 -25232.334,E2 -25232.334} C_VEL
LIN {X 0,Y 141.261,Z 279.959,A -85,B 0,C 180,E1 -25233.18,E2 -25233.18} C_VEL
LIN {X 0,Y 144.642,Z 284.743,A -85,B 0,C 180,E1 -25235.346,E2 -25235.346} C_VEL
LIN {X 0,Y 148.77,Z 291.204,A -85,B 0,C 180,E1 -25237.781,E2 -25237.781} C_VEL
LIN {X 0,Y 153.93,Z 301.833,A -85,B 0,C 180,E1 -25240.669,E2 -25240.669} C_VEL
LIN {X 0,Y 158.249,Z 312.739,A -85,B 0,C 180,E1 -25242.962,E2 -25242.962} C_VEL
LIN {X 0,Y 160.505,Z 319.52,A -85,B 0,C 180,E1 -25244.143,E2 -25244.143} C_VEL
LIN {X 0,Y 160.686,Z 325.006,A -85,B 0,C 180,E1 -25244.53,E2 -25244.53} C_VEL
LIN {X 0,Y 157.726,Z 367.98,A -85,B 0,C 180,E1 -25246.229,E2 -25246.229} C_VEL
LIN {X 0,Y 155.892,Z 381.234,A -85,B 0,C 180,E1 -25247.164,E2 -25247.164} C_VEL
LIN {X 0,Y 153.527,Z 393.045,A -85,B 0,C 180,E1 -25248.412,E2 -25248.412} C_VEL
LIN {X 0,Y 150.557,Z 404.456,A -85,B 0,C 180,E1 -25250.07,E2 -25250.07} C_VEL
LIN {X 0,Y 146.851,Z 416.199,A -85,B 0,C 180,E1 -25252.397,E2 -25252.397} C_VEL
LIN {X 0,Y 142.911,Z 426.737,A -85,B 0,C 180,E1 -25255.132,E2 -25255.132} C_VEL
LIN {X 0,Y 139.398,Z 435.351,A -85,B 0,C 180,E1 -25258.037,E2 -25258.037} C_VEL
LIN {X 0,Y 136.271,Z 442.849,A -85,B 0,C 180,E1 -25261.253,E2 -25261.253} C_VEL
LIN {X 0,Y 133.258,Z 449.884,A -85,B 0,C 180,E1 -25265.044,E2 -25265.044} C_VEL
LIN {X 0,Y 130.402,Z 456.349,A -85,B 0,C 180,E1 -25269.493,E2 -25269.493} C_VEL
LIN {X 0,Y 128.303,Z 461.474,A -85,B 0,C 180,E1 -25274.105,E2 -25274.105} C_VEL
LIN {X 0,Y 127.063,Z 465.45,A -85,B 0,C 180,E1 -25278.838,E2 -25278.838} C_VEL
LIN {X 0,Y 126.46,Z 468.378,A -85,B 0,C 180,E1 -25283.619,E2 -25283.619} C_VEL
LIN {X 0,Y 126.378,Z 469.761,A -85,B 0,C 180,E1 -25286.812,E2 -25286.812} C_VEL
LIN {X 0,Y 126.445,Z 470.741,A -85,B 0,C 180,E1 -25290,E2 -25290} C_VEL
LIN {X 0,Y 126.375,Z 471.318,A -85,B 0,C 180,E1 -25293.188,E2 -25293.188} C_VEL
LIN {X 0,Y 126.464,Z 471.497,A -85,B 0,C 180,E1 -25296.381,E2 -25296.381} C_VEL
LIN {X 0,Y 127.505,Z 470.615,A -85,B 0,C 180,E1 -25302.737,E2 -25302.737} C_VEL
LIN {X 0,Y 128.546,Z 469.6,A -85,B 0,C 180,E1 -25305.865,E2 -25305.865} C_VEL
LIN {X 0,Y 130.085,Z 467.948,A -85,B 0,C 180,E1 -25309.338,E2 -25309.338} C_VEL
LIN {X 0,Y 130.924,Z 466.48,A -85,B 0,C 180,E1 -25311.813,E2 -25311.813} C_VEL
LIN {X 0,Y 131.101,Z 463.57,A -85,B 0,C 180,E1 -25315.963,E2 -25315.963} C_VEL
LIN {X 0,Y 131.498,Z 460.86,A -85,B 0,C 180,E1 -25319.22,E2 -25319.22} C_VEL
LIN {X 0,Y 132.694,Z 458.467,A -85,B 0,C 180,E1 -25321.509,E2 -25321.509} C_VEL
LIN {X 0,Y 133.353,Z 457.578,A -85,B 0,C 180,E1 -25322.215,E2 -25322.215} C_VEL
LIN {X 0,Y 138.718,Z 450.988,A -85,B 0,C 180,E1 -25326.534,E2 -25326.534} C_VEL
LIN {X 0,Y 144.413,Z 443.422,A -85,B 0,C 180,E1 -25330.153,E2 -25330.153} C_VEL
LIN {X 0,Y 149.692,Z 435.697,A -85,B 0,C 180,E1 -25332.904,E2 -25332.904} C_VEL
LIN {X 0,Y 155.763,Z 425.219,A -85,B 0,C 180,E1 -25335.748,E2 -25335.748} C_VEL
LIN {X 0,Y 161.093,Z 414.568,A -85,B 0,C 180,E1 -25337.873,E2 -25337.873} C_VEL
LIN {X 0,Y 165.419,Z 404.268,A -85,B 0,C 180,E1 -25339.415,E2 -25339.415} C_VEL
LIN {X 0,Y 169.502,Z 391.966,A -85,B 0,C 180,E1 -25340.79,E2 -25340.79} C_VEL
LIN {X 0,Y 172.699,Z 379.025,A -85,B 0,C 180,E1 -25341.808,E2 -25341.808} C_VEL
LIN {X 0,Y 174.797,Z 366.844,A -85,B 0,C 180,E1 -25342.412,E2 -25342.412} C_VEL
LIN {X 0,Y 176.819,Z 342.042,A -85,B 0,C 180,E1 -25343.304,E2 -25343.304} C_VEL
LIN {X 0,Y 173.394,Z 332.832,A -85,B 0,C 180,E1 -25345.723,E2 -25345.723} C_VEL
LIN {X 0,Y 169.533,Z 323.837,A -85,B 0,C 180,E1 -25348.679,E2 -25348.679} C_VEL
LIN {X 0,Y 165.716,Z 316.023,A -85,B 0,C 180,E1 -25351.961,E2 -25351.961} C_VEL
LIN {X 0,Y 163.137,Z 311.159,A -85,B 0,C 180,E1 -25354.482,E2 -25354.482} C_VEL
LIN {X 0,Y 161.656,Z 308.831,A -85,B 0,C 180,E1 -25356.041,E2 -25356.041} C_VEL
LIN {X 0,Y 158.778,Z 304.654,A -85,B 0,C 180,E1 -25359.489,E2 -25359.489} C_VEL
LIN {X 0,Y 156.421,Z 301.403,A -85,B 0,C 180,E1 -25362.999,E2 -25362.999} C_VEL
LIN {X 0,Y 155.734,Z 300.096,A -85,B 0,C 180,E1 -25364.29,E2 -25364.29} C_VEL
LIN {X 0,Y 153.431,Z 297.455,A -85,B 0,C 180,E1 -25369.675,E2 -25369.675} C_VEL
LIN {X 0,Y 152.813,Z 294.911,A -85,B 0,C 180,E1 -25373.066,E2 -25373.066} C_VEL
LIN {X 0,Y 152.813,Z 294.841,A -85,B 0,C 180,E1 -25381.318,E2 -25381.318} C_VEL
LIN {X 0,Y 154.24,Z 298.502,A -85,B 0,C 180,E1 -25387.034,E2 -25387.034} C_VEL
LIN {X 0,Y 156.056,Z 300.443,A -85,B 0,C 180,E1 -25390.706,E2 -25390.706} C_VEL
LIN {X 0,Y 158.416,Z 304.157,A -85,B 0,C 180,E1 -25394.451,E2 -25394.451} C_VEL
LIN {X 0,Y 159.353,Z 305.39,A -85,B 0,C 180,E1 -25395.672,E2 -25395.672} C_VEL
LIN {X 0,Y 162.477,Z 310.048,A -85,B 0,C 180,E1 -25399.258,E2 -25399.258} C_VEL
LIN {X 0,Y 165.465,Z 314.683,A -85,B 0,C 180,E1 -25402.146,E2 -25402.146} C_VEL
LIN {X 0,Y 169.213,Z 320.76,A -85,B 0,C 180,E1 -25405.279,E2 -25405.279} C_VEL
LIN {X 0,Y 173.876,Z 329.257,A -85,B 0,C 180,E1 -25408.685,E2 -25408.685} C_VEL
LIN {X 0,Y 177.183,Z 336.126,A -85,B 0,C 180,E1 -25410.875,E2 -25410.875} C_VEL
LIN {X 0,Y 177.322,Z 336.551,A -85,B 0,C 180,E1 -25410.973,E2 -25410.973} C_VEL
LIN {X 0,Y 174.965,Z 362.903,A -85,B 0,C 180,E1 -25411.88,E2 -25411.88} C_VEL
LIN {X 0,Y 172.798,Z 375.617,A -85,B 0,C 180,E1 -25412.631,E2 -25412.631} C_VEL
LIN {X 0,Y 169.854,Z 387.638,A -85,B 0,C 180,E1 -25413.693,E2 -25413.693} C_VEL
LIN {X 0,Y 166.193,Z 398.656,A -85,B 0,C 180,E1 -25414.982,E2 -25414.982} C_VEL
LIN {X 0,Y 161.938,Z 409.03,A -85,B 0,C 180,E1 -25416.593,E2 -25416.593} C_VEL
LIN {X 0,Y 157.188,Z 418.862,A -85,B 0,C 180,E1 -25418.611,E2 -25418.611} C_VEL
LIN {X 0,Y 151.801,Z 428.469,A -85,B 0,C 180,E1 -25421.207,E2 -25421.207} C_VEL
LIN {X 0,Y 146.441,Z 436.479,A -85,B 0,C 180,E1 -25423.955,E2 -25423.955} C_VEL
LIN {X 0,Y 140.666,Z 444.301,A -85,B 0,C 180,E1 -25427.585,E2 -25427.585} C_VEL
LIN {X 0,Y 135.509,Z 450.532,A -85,B 0,C 180,E1 -25431.511,E2 -25431.511} C_VEL
LIN {X 0,Y 130.993,Z 455.466,A -85,B 0,C 180,E1 -25435.713,E2 -25435.713} C_VEL
LIN {X 0,Y 127.135,Z 459.257,A -85,B 0,C 180,E1 -25440.164,E2 -25440.164} C_VEL
LIN {X 0,Y 123.904,Z 462.148,A -85,B 0,C 180,E1 -25445.169,E2 -25445.169} C_VEL
LIN {X 0,Y 121.716,Z 463.799,A -85,B 0,C 180,E1 -25449.73,E2 -25449.73} C_VEL
LIN {X 0,Y 119.77,Z 464.746,A -85,B 0,C 180,E1 -25456.425,E2 -25456.425} C_VEL
LIN {X 0,Y 119.337,Z 464.639,A -85,B 0,C 180,E1 -25459.824,E2 -25459.824} C_VEL
LIN {X 0,Y 119.214,Z 464.101,A -85,B 0,C 180,E1 -25463.229,E2 -25463.229} C_VEL
LIN {X 0,Y 119.488,Z 462.18,A -85,B 0,C 180,E1 -25469.242,E2 -25469.242} C_VEL
LIN {X 0,Y 120.429,Z 459.079,A -85,B 0,C 180,E1 -25475.022,E2 -25475.022} C_VEL
LIN {X 0,Y 121.952,Z 455.298,A -85,B 0,C 180,E1 -25479.956,E2 -25479.956} C_VEL
LIN {X 0,Y 124.219,Z 450.4,A -85,B 0,C 180,E1 -25484.75,E2 -25484.75} C_VEL
LIN {X 0,Y 127.165,Z 444.244,A -85,B 0,C 180,E1 -25489.366,E2 -25489.366} C_VEL
LIN {X 0,Y 130.925,Z 436.562,A -85,B 0,C 180,E1 -25493.741,E2 -25493.741} C_VEL
LIN {X 0,Y 135.224,Z 426.942,A -85,B 0,C 180,E1 -25497.889,E2 -25497.889} C_VEL
LIN {X 0,Y 139.375,Z 417,A -85,B 0,C 180,E1 -25501.122,E2 -25501.122} C_VEL
LIN {X 0,Y 143.331,Z 405.759,A -85,B 0,C 180,E1 -25503.901,E2 -25503.901} C_VEL
LIN {X 0,Y 146.626,Z 394.75,A -85,B 0,C 180,E1 -25505.956,E2 -25505.956} C_VEL
LIN {X 0,Y 149.529,Z 382.545,A -85,B 0,C 180,E1 -25507.663,E2 -25507.663} C_VEL
LIN {X 0,Y 151.755,Z 369.687,A -85,B 0,C 180,E1 -25508.904,E2 -25508.904} C_VEL
LIN {X 0,Y 153.263,Z 356.202,A -85,B 0,C 180,E1 -25509.701,E2 -25509.701} C_VEL
LIN {X 0,Y 155.998,Z 316.777,A -85,B 0,C 180,E1 -25511.232,E2 -25511.232} C_VEL
LIN {X 0,Y 150.98,Z 306.36,A -85,B 0,C 180,E1 -25513.852,E2 -25513.852} C_VEL
LIN {X 0,Y 146.068,Z 297.679,A -85,B 0,C 180,E1 -25516.619,E2 -25516.619} C_VEL
LIN {X 0,Y 141.508,Z 290.521,A -85,B 0,C 180,E1 -25519.453,E2 -25519.453} C_VEL
LIN {X 0,Y 137.153,Z 284.194,A -85,B 0,C 180,E1 -25522.489,E2 -25522.489} C_VEL
LIN {X 0,Y 134.172,Z 280.072,A -85,B 0,C 180,E1 -25524.817,E2 -25524.817} C_VEL
LIN {X 0,Y 131.498,Z 276.721,A -85,B 0,C 180,E1 -25527.103,E2 -25527.103} C_VEL
LIN {X 0,Y 130.653,Z 275.35,A -85,B 0,C 180,E1 -25527.914,E2 -25527.914} C_VEL
LIN {X 0,Y 128.153,Z 272.943,A -85,B 0,C 180,E1 -25530.312,E2 -25530.312} C_VEL
LIN {X 0,Y 126.732,Z 270.086,A -85,B 0,C 180,E1 -25532.012,E2 -25532.012} C_VEL
LIN {X 0,Y 123.843,Z 268.252,A -85,B 0,C 180,E1 -25535.38,E2 -25535.38} C_VEL
LIN {X 0,Y 122.504,Z 266.008,A -85,B 0,C 180,E1 -25537.427,E2 -25537.427} C_VEL
LIN {X 0,Y 122.053,Z 264.231,A -85,B 0,C 180,E1 -25538.503,E2 -25538.503} C_VEL
LIN {X 0,Y 122.109,Z 264.269,A -85,B 0,C 180,E1 -25543.275,E2 -25543.275} C_VEL
LIN {X 0,Y 122.312,Z 264.192,A -85,B 0,C 180,E1 -25547.637,E2 -25547.637} C_VEL
LIN {X 0,Y 122.416,Z 264.222,A -85,B 0,C 180,E1 -25553.406,E2 -25553.406} C_VEL
LIN {X 0,Y 123.04,Z 264.153,A -85,B 0,C 180,E1 -25560,E2 -25560} C_VEL
LIN {X 0,Y 122.451,Z 264.231,A -85,B 0,C 180,E1 -25566.591,E2 -25566.591} C_VEL
LIN {X 0,Y 122.446,Z 264.211,A -85,B 0,C 180,E1 -25569.915,E2 -25569.915} C_VEL
LIN {X 0,Y 122.141,Z 264.346,A -85,B 0,C 180,E1 -25575.433,E2 -25575.433} C_VEL
LIN {X 0,Y 122.868,Z 266.779,A -85,B 0,C 180,E1 -25576.832,E2 -25576.832} C_VEL
LIN {X 0,Y 124.838,Z 269.073,A -85,B 0,C 180,E1 -25579.527,E2 -25579.527} C_VEL
